(*=======================================================*)
	20:
		IF fb_state_entry.E THEN
			haspel1_ctrl_out.b_init := TRUE;
			haspel2_ctrl_out.b_init := TRUE;
			haspel3_ctrl_out.b_init := TRUE;
			haspel4_ctrl_out.b_init := TRUE;
		END_IF
		(*-----------------------Weiterschaltbedingungen----------------------------*)
		IF  	haspel1_ctrl_in.b_bereit AND
			haspel2_ctrl_in.b_bereit AND
			haspel3_ctrl_in.b_bereit AND
			haspel4_ctrl_in.b_bereit
			THEN
				haspel1_ctrl_out.b_init := FALSE;
				haspel2_ctrl_out.b_init := FALSE;
				haspel3_ctrl_out.b_init := FALSE;
				haspel4_ctrl_out.b_init := FALSE;
				fb_tof_motor.IN := TRUE;
				fb_state_entry.i16_next_step := BEREIT;
		END_IF

(*=======================================================*)
	BEREIT: (* Haspelmotor läuft *)
		IF fb_state_entry.E THEN
			st_ctrl_out.b_bereit := TRUE;
		END_IF

		a_motor_drehrichtung_links 	:= e_druckwaechter AND fb_tof_motor.Q AND b_drehrichtung_antrieb_links;
		a_motor_drehrichtung_rechts := e_druckwaechter AND fb_tof_motor.Q AND NOT b_drehrichtung_antrieb_links;

		(* Abschaltzeit für Haspelmotor nachtriggern*)
		IF 	haspel1_ctrl_in.b_kontroller_start OR
			haspel2_ctrl_in.b_kontroller_start OR
			haspel3_ctrl_in.b_kontroller_start OR
			haspel4_ctrl_in.b_kontroller_start
			THEN
				fb_tof_motor.IN := TRUE;
		ELSE
			fb_tof_motor.IN := FALSE;
		END_IF

(*=======================================================*)
	FEHLER:
		IF fb_state_entry.E THEN
			fb_ton_quitt.IN := FALSE;
			st_ctrl_out.b_fehler := TRUE;
			haspel1_ctrl_out.b_stop := FALSE;
			haspel2_ctrl_out.b_stop := FALSE;
			haspel3_ctrl_out.b_stop := FALSE;
			haspel4_ctrl_out.b_stop := FALSE;
			haspel1_ctrl_out.b_quitt := FALSE;
			haspel2_ctrl_out.b_quitt := FALSE;
			haspel3_ctrl_out.b_quitt := FALSE;
			haspel4_ctrl_out.b_quitt := FALSE;
			a_motor_drehrichtung_links 	:= FALSE;
			a_motor_drehrichtung_rechts := FALSE;
		END_IF

		(*-----------------------Weiterschaltbedingungen----------------------------*)
		IF st_ctrl_in.b_quitt AND NOT fb_state_entry.E THEN
			haspel1_ctrl_out.b_quitt := TRUE;
			haspel2_ctrl_out.b_quitt := TRUE;
			haspel3_ctrl_out.b_quitt := TRUE;
			haspel4_ctrl_out.b_quitt := TRUE;
			st_ctrl_out.b_fehler := FALSE;
			fb_ton_quitt.IN := TRUE;
		END_IF

		IF fb_ton_quitt.Q THEN
			fb_ton_quitt.IN := FALSE;
			fb_state_entry.i16_next_step := INIT;
		END_IF

(*=======================================================*)
	STOP:
		IF fb_state_entry.E THEN
			a_motor_drehrichtung_links 	:= FALSE;
			a_motor_drehrichtung_rechts := FALSE;
			haspel1_ctrl_out.b_stop := TRUE;
			haspel2_ctrl_out.b_stop := TRUE;
			haspel3_ctrl_out.b_stop := TRUE;
			haspel4_ctrl_out.b_stop := TRUE;
			haspel1_ctrl_out.b_quitt := FALSE;
			haspel2_ctrl_out.b_quitt := FALSE;
			haspel3_ctrl_out.b_quitt := FALSE;
			haspel4_ctrl_out.b_quitt := FALSE;
			fb_ton_quitt.IN := FALSE;
		END_IF

		(*-----------------------Weiterschaltbedingungen----------------------------*)
		IF st_ctrl_in.b_quitt AND NOT fb_state_entry.E THEN
			haspel1_ctrl_out.b_stop := FALSE;
			haspel2_ctrl_out.b_stop := FALSE;
			haspel3_ctrl_out.b_stop := FALSE;
			haspel4_ctrl_out.b_stop := FALSE;
			haspel1_ctrl_out.b_quitt := TRUE;
			haspel2_ctrl_out.b_quitt := TRUE;
			haspel3_ctrl_out.b_quitt := TRUE;
			haspel4_ctrl_out.b_quitt := TRUE;

			fb_ton_quitt.IN := TRUE;
		END_IF

		IF fb_ton_quitt.Q THEN
			fb_ton_quitt.IN := FALSE;
			fb_state_entry.i16_next_step := INIT;
		END_IF
END_CASE

fb_state_entry(
	i16_next_step:= , 
	i16_pos:= 2,
	s_debugtext:= ,
	E=> , 
	X=> , 
	i16_step=> ,
	i16_last_step=> );

IF st_config.b_config_fertig THEN
	(* Fehlermeldungen und Betriebsmeldungen ab dem Startindex in die globalen Meldungsarrays schreiben *)
	garr_stoermeldungen[st_config.i16_meld_startindex + 0] := FALSE;
	garr_stoermeldungen[st_config.i16_meld_startindex + 1] := FALSE;
	garr_stoermeldungen[st_config.i16_meld_startindex + 2] := FALSE;
	garr_stoermeldungen[st_config.i16_meld_startindex + 3] := FALSE;
	garr_stoermeldungen[st_config.i16_meld_startindex + 4] := FALSE;
	garr_stoermeldungen[st_config.i16_meld_startindex + 5] := FALSE;
	garr_stoermeldungen[st_config.i16_meld_startindex + 6] := FALSE;
	garr_stoermeldungen[st_config.i16_meld_startindex + 7] := FALSE;
	garr_stoermeldungen[st_config.i16_meld_startindex + 8] := FALSE;
	garr_stoermeldungen[st_config.i16_meld_startindex + 9] := FALSE;
	garr_stoermeldungen[st_config.i16_meld_startindex + 10] := FALSE;
	garr_stoermeldungen[st_config.i16_meld_startindex + 11] := FALSE;
	garr_stoermeldungen[st_config.i16_meld_startindex + 12] := FALSE;
	garr_stoermeldungen[st_config.i16_meld_startindex + 13] := FALSE;
	garr_stoermeldungen[st_config.i16_meld_startindex + 14] := FALSE;
	garr_stoermeldungen[st_config.i16_meld_startindex + 15] := FALSE;
	garr_stoermeldungen[st_config.i16_meld_startindex + 16] := FALSE;
	garr_stoermeldungen[st_config.i16_meld_startindex + 17] := FALSE;
	garr_stoermeldungen[st_config.i16_meld_startindex + 18] := FALSE;
	garr_stoermeldungen[st_config.i16_meld_startindex + 19] := FALSE;
	
	garr_betriebsmeldungen[st_config.i16_meld_startindex + 0] := FALSE;
	garr_betriebsmeldungen[st_config.i16_meld_startindex + 1] := FALSE;
	garr_betriebsmeldungen[st_config.i16_meld_startindex + 2] := FALSE;
	garr_betriebsmeldungen[st_config.i16_meld_startindex + 3] := FALSE;
	garr_betriebsmeldungen[st_config.i16_meld_startindex + 4] := FALSE;
	garr_betriebsmeldungen[st_config.i16_meld_startindex + 5] := FALSE;
	garr_betriebsmeldungen[st_config.i16_meld_startindex + 6] := FALSE;
	garr_betriebsmeldungen[st_config.i16_meld_startindex + 7] := FALSE;
	garr_betriebsmeldungen[st_config.i16_meld_startindex + 8] := FALSE;
	garr_betriebsmeldungen[st_config.i16_meld_startindex + 9] := FALSE;
	garr_betriebsmeldungen[st_config.i16_meld_startindex + 10] := FALSE;
	garr_betriebsmeldungen[st_config.i16_meld_startindex + 11] := FALSE;
	garr_betriebsmeldungen[st_config.i16_meld_startindex + 12] := FALSE;
	garr_betriebsmeldungen[st_config.i16_meld_startindex + 13] := FALSE;
	garr_betriebsmeldungen[st_config.i16_meld_startindex + 14] := FALSE;
	garr_betriebsmeldungen[st_config.i16_meld_startindex + 15] := FALSE;
	garr_betriebsmeldungen[st_config.i16_meld_startindex + 16] := FALSE;
	garr_betriebsmeldungen[st_config.i16_meld_startindex + 17] := FALSE;
	garr_betriebsmeldungen[st_config.i16_meld_startindex + 18] := FALSE;
	garr_betriebsmeldungen[st_config.i16_meld_startindex + 19] := FALSE;
END_IF
END_PROGRAM

(* POU EPT Lib/Programmbausteine/Routing/PC-Suche/ST_RoutingNachbarPC, ST *)
PROGRAM ST_RoutingNachbarPC
VAR_INPUT
	st_config						: struct_config;
	st_ctrl_in						: struct_ctrl_in;
END_VAR
VAR_OUTPUT
	st_ctrl_out					: struct_ctrl_out;
END_VAR
VAR
	arr_read_routing_info			: ARRAY [0..31] OF ST_AmsRouteEntry;
	fb_add_route_entry			: FB_AddRouteEntry;
	fb_enum_route_entry			: FB_EnumRouteEntry;
	fb_ton_quitt					: TON;
	fb_state_entry					: ST_StateEntry;
	i16_geschriebene_eintraege	: INT := 0;
	i16_vorhandene_eintraege		: INT := 0;
	b_ibn_start_routing			: BOOL := FALSE;
	fb_r_trig_ibn_start_routing		: R_TRIG;
	fb_ton_ibn_start_routing		: TON;
	sm_fehler_remotesuche		: BOOL := FALSE;
	sm_fehler_netid				: BOOL := FALSE;
	fb_suche_remote_pc			: ST_SucheRemotePC;
	fb_get_local_ams_netid		: ST_GetLocalAMSNetID;
	i16_eintrag					: INT := 0;
END_VAR
fb_ton_quitt(IN:= , PT:= t#100ms, Q=> , ET=> );
fb_r_trig_ibn_start_routing(CLK:= b_ibn_start_routing, Q=> );
fb_ton_ibn_start_routing(IN:= , PT:= t#1s, Q=> , ET=> );

IF fb_r_trig_ibn_start_routing.Q THEN
	fb_ton_ibn_start_routing.IN := TRUE;
ELSE
	IF fb_ton_ibn_start_routing.Q THEN
		b_ibn_start_routing := FALSE;
	 	fb_ton_ibn_start_routing.IN := FALSE;
	END_IF
END_IF

fb_state_entry(
	i16_next_step:= ,
	i16_pos:= 1,
	s_debugtext:= ,
	E=> ,
	X=> ,
	i16_step=> ,
	i16_last_step=> );

CASE fb_state_entry.i16_step OF
(*=======================================================*)
	0:	(* Initialisierung *)
		st_ctrl_out.b_fehler := TRUE;
		st_ctrl_out.b_bereit := TRUE;
		st_ctrl_out.b_fertig := TRUE;
		fb_add_route_entry.bExecute := FALSE;
		fb_enum_route_entry.bExecute := FALSE;
		fb_suche_remote_pc.bQuit := FALSE;
		fb_suche_remote_pc.bExecute := FALSE;
		fb_get_local_ams_netid .bQuit := FALSE;
		fb_get_local_ams_netid.bExecute := FALSE;
		fb_enum_route_entry.eCmd := eEnumCmd_First;
		i16_geschriebene_eintraege := 0;
		i16_vorhandene_eintraege := 0;
		sm_fehler_remotesuche := FALSE;
		sm_fehler_netid := FALSE;

		FOR i16_eintrag := 0  TO (SIZEOF (arr_read_routing_info) / SIZEOF (arr_read_routing_info[0])) BY 1DO
			arr_read_routing_info[i16_eintrag].sName := '';
			arr_read_routing_info[i16_eintrag].sNetID := '';
			arr_read_routing_info[i16_eintrag].sAddress := '';
			arr_read_routing_info[i16_eintrag].eTransport := eRouteTransport_TCP_IP;
		END_FOR

		fb_state_entry.i16_next_step := 10;

(*=======================================================*)
	10:	(* Die AMS-NetID des lokalen PC ermitteln *)
		IF fb_state_entry.E THEN
			fb_get_local_ams_netid.bExecute := TRUE;
		END_IF

		IF fb_get_local_ams_netid.bBusy THEN
			fb_get_local_ams_netid.bExecute := FALSE;
			fb_state_entry.i16_next_step := 20;
		END_IF

(*=======================================================*)
	20:
		IF NOT fb_get_local_ams_netid.bBusy  THEN
			IF NOT fb_get_local_ams_netid.bError THEN
				fb_state_entry.i16_next_step := 100;
			ELSE	(* Fehler *)
				sm_fehler_netid := TRUE;
				fb_state_entry.i16_next_step := 1000;
			END_IF
		END_IF

(*=======================================================*)
	100:	(* Ersten Routing Eintrag im Routingtable lesen *)
		IF fb_state_entry.E THEN
			fb_enum_route_entry.bExecute := TRUE;
		END_IF

		IF fb_enum_route_entry.bBusy THEN
			fb_enum_route_entry.bExecute := FALSE;
			fb_state_entry.i16_next_step := 110;
		END_IF

(*=======================================================*)
	110:	(* Routinginformation ist vorhanden *)
		IF NOT fb_enum_route_entry.bBusy  THEN
			IF NOT fb_enum_route_entry.bError THEN
				IF NOT fb_enum_route_entry.bEOE THEN
					arr_read_routing_info[i16_vorhandene_eintraege] := fb_enum_route_entry.stRoute;
					fb_enum_route_entry.eCmd := eEnumCmd_Next;
					fb_state_entry.i16_next_step := 120;
				ELSE	(* Alle vorhandenen Routingeinträge  wurden eingelesen*)
					fb_state_entry.i16_next_step := 130;
				END_IF
			ELSE	(* Fehler *)
				fb_state_entry.i16_next_step := 1000;
			END_IF
		END_IF

(*=======================================================*)
	120:	(* Zähler erhöhen *)
		IF fb_state_entry.E THEN
			i16_vorhandene_eintraege := i16_vorhandene_eintraege + 1;
		END_IF

		fb_state_entry.i16_next_step := 100;

(*=======================================================*)
	130:	(* Suche Nachbar-PCs im Maschinennetz *)
		IF fb_state_entry.E THEN
			fb_suche_remote_pc.bExecute := TRUE;
		END_IF

		IF fb_suche_remote_pc.bBusy THEN
			fb_suche_remote_pc.bExecute := FALSE;
			fb_state_entry.i16_next_step := 140;
		END_IF

(*=======================================================*)
	140:	(* Suchvorgang und beendet *)
		IF NOT fb_suche_remote_pc.bBusy  THEN
			IF NOT fb_suche_remote_pc.bError THEN
				fb_state_entry.i16_next_step := 150;
			ELSE	(* Fehler *)
				sm_fehler_remotesuche := TRUE;
				fb_state_entry.i16_next_step := 1000;
			END_IF
		END_IF

(*=======================================================*)
	150:	(* Die Route der gefundenen Nachbar-PCs eintragen *)
		IF fb_state_entry.E THEN
			fb_add_route_entry.stRoute.sName := fb_suche_remote_pc.st_remote_pcinfo_struct[i16_geschriebene_eintraege].Name;
			fb_add_route_entry.stRoute.sNetID := fb_suche_remote_pc.st_remote_pcinfo_struct[i16_geschriebene_eintraege].NetId;
			fb_add_route_entry.stRoute.sAddress := DELETE(fb_add_route_entry.stRoute.sNetID, 4, 12);
			fb_add_route_entry.stRoute.eTransport := eRouteTransport_TCP_IP;
			fb_add_route_entry.bExecute :=TRUE;
			i16_geschriebene_eintraege := i16_geschriebene_eintraege + 1;
		END_IF

		IF fb_add_route_entry.bBusy THEN
			fb_add_route_entry.bExecute := FALSE;
			fb_state_entry.i16_next_step := 160;
		END_IF

(*=======================================================*)
	160:	(* Routingtable füllen läuft *)
		IF NOT fb_add_route_entry.bBusy THEN
			IF NOT fb_add_route_entry.bError THEN	(* Route wurde erfolgreich hinzugefügt *)
				(* Routingtable mit fehlenden Stationsadressen füllen wenn notwendig *)
				IF i16_geschriebene_eintraege < i16_vorhandene_eintraege THEN
					fb_state_entry.i16_next_step := 150;
				ELSE
					fb_state_entry.i16_next_step := 999;
				END_IF
			ELSE	(* Fehler *)
				fb_state_entry.i16_next_step := 1000;
			END_IF
		END_IF

(*=======================================================*)
	999: (* Ende: Alle Stationen wurden im Routingtable eingetragen *)
		IF fb_state_entry.E THEN
			st_ctrl_out.b_fertig := TRUE;
		END_IF

(*=======================================================*)
	1000: (* Fehler *)
		IF fb_state_entry.E THEN
			st_ctrl_out.b_fehler := TRUE;
			fb_ton_quitt.IN := FALSE;
			fb_add_route_entry.bExecute := FALSE;
			fb_enum_route_entry.bExecute := FALSE;
			fb_suche_remote_pc.bExecute := FALSE;
			fb_suche_remote_pc.bQuit := FALSE;
			fb_get_local_ams_netid.bExecute := FALSE;
			fb_get_local_ams_netid.bQuit := FALSE;
		END_IF

		(*-----------------------Weiterschaltbedingungen----------------------------*)
		IF st_ctrl_in.b_quitt AND NOT fb_state_entry.E THEN
			st_ctrl_out.b_fehler := FALSE;
			fb_ton_quitt.IN := TRUE;
			fb_suche_remote_pc.bQuit := TRUE;
			fb_get_local_ams_netid .bQuit := TRUE;
		END_IF

		IF fb_ton_quitt.Q OR  fb_r_trig_ibn_start_routing.Q THEN
			fb_ton_quitt.IN := FALSE;
			fb_state_entry.i16_next_step := 0;
		END_IF
END_CASE

fb_state_entry(
	i16_next_step:= , 
	i16_pos:= 2,
	s_debugtext:= ,
	E=> ,
	X=> , 
	i16_step=> ,
	i16_last_step=> );

fb_get_local_ams_netid(
	bExecute:= , 
	bQuit:= , 
	bBusy=> , 
	bReady=> , 
	bError=> , 
	nErrId=> , 
	s_ams_netid=> );

fb_suche_remote_pc(
	bExecute:= ,
	bQuit:= , 
	bBusy=> , 
	bError=> , 
	nErrId=> );

fb_add_route_entry(
	sNetID:= ,
	stRoute:= ,
	bExecute:= ,
	tTimeout:= DEFAULT_ADS_TIMEOUT,
	bBusy=> , 
	bError=> , 
	nErrID=> );

fb_enum_route_entry(
	sNetID:= ,
	eCmd:= , 
	bExecute:= , 
	tTimeout:= DEFAULT_ADS_TIMEOUT,
	bBusy=> , 
	bError=> , 
	nErrID=> , 
	bEOE=> , 
	stRoute=> );

IF st_config.b_config_fertig THEN
	garr_stoermeldungen[st_config.i16_meld_startindex + 0] := sm_fehler_remotesuche;
	garr_stoermeldungen[st_config.i16_meld_startindex + 1] := sm_fehler_netid;
	garr_stoermeldungen[st_config.i16_meld_startindex + 2] := FALSE;
	garr_stoermeldungen[st_config.i16_meld_startindex + 3] := FALSE;
	garr_stoermeldungen[st_config.i16_meld_startindex + 4] := FALSE;
	garr_stoermeldungen[st_config.i16_meld_startindex + 5] := FALSE;
	garr_stoermeldungen[st_config.i16_meld_startindex + 6] := FALSE;
	garr_stoermeldungen[st_config.i16_meld_startindex + 7] := FALSE;
	garr_stoermeldungen[st_config.i16_meld_startindex + 8] := FALSE;
	garr_stoermeldungen[st_config.i16_meld_startindex + 9] := FALSE;
	garr_stoermeldungen[st_config.i16_meld_startindex + 10] := FALSE;
	garr_stoermeldungen[st_config.i16_meld_startindex + 11] := FALSE;
	garr_stoermeldungen[st_config.i16_meld_startindex + 12] := FALSE;
	garr_stoermeldungen[st_config.i16_meld_startindex + 13] := FALSE;
	garr_stoermeldungen[st_config.i16_meld_startindex + 14] := FALSE;
	garr_stoermeldungen[st_config.i16_meld_startindex + 15] := FALSE;
	garr_stoermeldungen[st_config.i16_meld_startindex + 16] := FALSE;
	garr_stoermeldungen[st_config.i16_meld_startindex + 17] := FALSE;
	garr_stoermeldungen[st_config.i16_meld_startindex + 18] := FALSE;
	garr_stoermeldungen[st_config.i16_meld_startindex + 19] := FALSE;
	
	garr_betriebsmeldungen[st_config.i16_meld_startindex + 0] := FALSE;
	garr_betriebsmeldungen[st_config.i16_meld_startindex + 1] := FALSE;
	garr_betriebsmeldungen[st_config.i16_meld_startindex + 2] := FALSE;
	garr_betriebsmeldungen[st_config.i16_meld_startindex + 3] := FALSE;
	garr_betriebsmeldungen[st_config.i16_meld_startindex + 4] := FALSE;
	garr_betriebsmeldungen[st_config.i16_meld_startindex + 5] := FALSE;
	garr_betriebsmeldungen[st_config.i16_meld_startindex + 6] := FALSE;
	garr_betriebsmeldungen[st_config.i16_meld_startindex + 7] := FALSE;
	garr_betriebsmeldungen[st_config.i16_meld_startindex + 8] := FALSE;
	garr_betriebsmeldungen[st_config.i16_meld_startindex + 9] := FALSE;
	garr_betriebsmeldungen[st_config.i16_meld_startindex + 10] := FALSE;
	garr_betriebsmeldungen[st_config.i16_meld_startindex + 11] := FALSE;
	garr_betriebsmeldungen[st_config.i16_meld_startindex + 12] := FALSE;
	garr_betriebsmeldungen[st_config.i16_meld_startindex + 13] := FALSE;
	garr_betriebsmeldungen[st_config.i16_meld_startindex + 14] := FALSE;
	garr_betriebsmeldungen[st_config.i16_meld_startindex + 15] := FALSE;
	garr_betriebsmeldungen[st_config.i16_meld_startindex + 16] := FALSE;
	garr_betriebsmeldungen[st_config.i16_meld_startindex + 17] := FALSE;
	garr_betriebsmeldungen[st_config.i16_meld_startindex + 18] := FALSE;
	garr_betriebsmeldungen[st_config.i16_meld_startindex + 19] := FALSE;
END_IF
END_PROGRAM

(* POU EPT Lib/Programmbausteine/Routing/PC-Suche/ST_SucheRemotePC, ST *)
FUNCTION_BLOCK ST_SucheRemotePC
VAR_INPUT
	bExecute			: BOOL;
	bQuit				: BOOL;
END_VAR
VAR_OUTPUT
	bBusy				: BOOL;
	bError				: BOOL;
	nErrId				: UDINT;
END_VAR
VAR
	fb_ton_quitt					: TON;
	fb_state_entry					: ST_StateEntry;
	fb_r_trig_execute				: R_TRIG;
	i							: INT := 0;
	b_ibn_start					: BOOL := FALSE;
	fb_r_trig_ibn_start				: R_TRIG;
	fb_ton_ibn_start				: TON;
	fb_get_remote_pcinfo			:GetRemotePCInfo;
	st_remote_pcinfo_struct		:REMOTEPCINFOSTRUCT;
							       (*TYPE REMOTEPCINFOSTRUCT
									ARRAY[0..99] OF REMOTEPC;
								END_TYPE*)
							      (*TYPE REMOTEPC
								STRUCT
									NetId 	: T_AmsNetId;
									Name 	: STRING(31);
								END_STRUCT
								END_TYPE*)
END_VAR
fb_r_trig_execute(CLK:= bExecute, Q=> );
fb_ton_quitt(IN:= , PT:= t#100ms, Q=> , ET=> );

fb_r_trig_ibn_start(CLK:= b_ibn_start, Q=> );
fb_ton_ibn_start(IN:= , PT:= t#1s, Q=> , ET=> );

IF fb_r_trig_ibn_start.Q THEN
	fb_ton_ibn_start.IN := TRUE;
ELSE
	IF fb_ton_ibn_start.Q THEN
		b_ibn_start := FALSE;
	 	fb_ton_ibn_start.IN := FALSE;
	END_IF
END_IF

fb_state_entry(
	i16_next_step:= ,
	i16_pos:= 1,
	s_debugtext:= ,
	E=> ,
	X=> , 
	i16_step=> ,
	i16_last_step=> );

CASE fb_state_entry.i16_step OF
(*=======================================================*)
	0:(* INIT *)
		bBusy := FALSE;
		bError := FALSE;
		nErrId := 0;
		fb_get_remote_pcinfo.START := FALSE;
		fb_state_entry.i16_next_step := 10;

(*=======================================================*)
	10:	(* Warte auf Execute-Befehl *)
		IF fb_state_entry.E THEN
			bBusy := FALSE;
		END_IF

		IF fb_r_trig_execute.Q OR fb_r_trig_ibn_start.Q THEN
			bBusy := TRUE;
			fb_state_entry.i16_next_step := 100;
		END_IF

(*=======================================================*)
	100:	(* Starte mit Auslesen der über ADS verbundenen Nachbar-PCs *)
		IF fb_state_entry.E THEN
			fb_get_remote_pcinfo.START := TRUE;
		END_IF

		IF fb_get_remote_pcinfo.BUSY THEN
			fb_get_remote_pcinfo.START := FALSE;
			fb_state_entry.i16_next_step := 110;
		END_IF

(*=======================================================*)
	110:	(* Routinginformation über die Nachbar-PCs ist vorhanden *)
		IF NOT fb_get_remote_pcinfo.BUSY  THEN
			IF NOT fb_get_remote_pcinfo.ERR THEN
				fb_state_entry.i16_next_step := 999;
			ELSE	(* Fehler *)
				fb_state_entry.i16_next_step := 1000;
			END_IF
		END_IF

(*=======================================================*)
	999:	(* Kontrollschritt: Nachbar-PC ist gefunden *)
		fb_state_entry.i16_next_step := 10;

(*=======================================================*)
	1000: (* Fehler *)
		IF fb_state_entry.E THEN
			bBusy := FALSE;
			bError := TRUE;
			fb_ton_quitt.IN := FALSE;
		END_IF

		(*-----------------------Weiterschaltbedingungen----------------------------*)
		IF bQuit AND NOT fb_state_entry.E THEN
			bError := FALSE;
			fb_ton_quitt.IN := TRUE;
		END_IF

		IF fb_ton_quitt.Q THEN
			fb_ton_quitt.IN := FALSE;
			fb_state_entry.i16_next_step := 0;
		END_IF
END_CASE

fb_state_entry(
	i16_next_step:= , 
	i16_pos:= 2,
	s_debugtext:= ,
	E=> ,
	X=> , 
	i16_step=> ,
	i16_last_step=> );

fb_get_remote_pcinfo(
	NETID:= , 
	START:= , 
	TMOUT:= , 
	BUSY=> , 
	ERR=> , 
	ERRID=> , 
	RemotePCInfo=> st_remote_pcinfo_struct);
END_FUNCTION_BLOCK

(* POU EPT Lib/Funktionen/BOOLARRAY_TO_BYTE, ST *)
FUNCTION BOOLARRAY_TO_BYTE : BYTE
VAR_INPUT
	p_adr_buffer			: POINTER TO ARRAY[0..7] OF BOOL;
END_VAR
VAR
	tmp_buffer			: ARRAY[0..7] OF BOOL;
	tmp_byte				: BYTE;
	i16_index			: INT;
END_VAR
(* Aus einem Boolarray, soll ein Byte entstehen *)
tmp_buffer := p_adr_buffer^;

tmp_byte := 2#0;

FOR i16_index := 7 TO 0 BY -1 DO
	tmp_byte := tmp_byte OR BOOL_TO_BYTE(tmp_buffer[i16_index]);
	IF i16_index > 0 THEN
		tmp_byte := SHL(tmp_byte, 1);
	END_IF
END_FOR;

BOOLARRAY_TO_BYTE := tmp_byte; (* Rückgabewert der Funktion *)
END_FUNCTION

(* POU EPT Lib/Funktionen/BOOLARRAY_TO_DWORD, ST *)
FUNCTION BOOLARRAY_TO_DWORD : DWORD
VAR_INPUT
	p_adr_buffer			: POINTER TO ARRAY[0..31] OF BOOL;
END_VAR
VAR
	tmp_buffer			: ARRAY[0..31] OF BOOL;
	tmp_dword			: DWORD;
	i16_index			: INT;
END_VAR
(* Aus einem Boolarray, soll ein Doppelword entstehen *)
tmp_buffer := p_adr_buffer^;

tmp_dword := 2#0;

FOR i16_index := 31 TO 0 BY -1 DO
	tmp_dword := tmp_dword OR BOOL_TO_DWORD(tmp_buffer[i16_index]);
	IF i16_index > 0 THEN
		tmp_dword := SHL(tmp_dword, 1);
	END_IF
END_FOR;

BOOLARRAY_TO_DWORD := tmp_dword; (* Rückgabewert der Funktion *)
END_FUNCTION

(* POU EPT Lib/Funktionen/BOOLARRAY_TO_WORD, ST *)
FUNCTION BOOLARRAY_TO_WORD : WORD
VAR_INPUT
	p_adr_buffer			: POINTER TO ARRAY[0..15] OF BOOL;
END_VAR
VAR
	tmp_buffer			: ARRAY[0..15] OF BOOL;
	tmp_word			: WORD;
	i16_index			: INT;
END_VAR
(* Aus einem Boolarray, soll ein Word entstehen *)
tmp_buffer := p_adr_buffer^;

tmp_word := 2#0;

FOR i16_index := 15 TO 0 BY -1 DO
	tmp_word := tmp_word OR BOOL_TO_WORD(tmp_buffer[i16_index]);
	IF i16_index > 0 THEN
		tmp_word := SHL(tmp_word, 1);
	END_IF
END_FOR;

BOOLARRAY_TO_WORD := tmp_word; (* Rückgabewert der Funktion *)
END_FUNCTION

(* POU EPT Lib/Funktionen/BYTEARRAY_TO_STRING_WITH_DELIMITER, ST *)
FUNCTION BYTEARRAY_TO_STRING_WITH_DELIMITER : STRING
VAR_INPUT
	p_adr_buffer			: POINTER TO ARRAY[0..100] OF BYTE;
	i16_buffer_laenge		: INT;
	str_delimiter			: STRING; (* Punkt zum trennen der einzelnen Zahlen in der Net-Adresse *)
END_VAR
VAR
	tmp_buffer			: ARRAY[0..100] OF BYTE;
	tmp_string			: STRING;
	i16_index			: INT;
END_VAR
(* Aus einem Bytearray, welches die einzelnen Zahlen der Net-Adresse beinhaltet wird ein String erzeugt, welcher die Zahlen getrennt durch Punkte enthält *)
tmp_buffer := p_adr_buffer^;

tmp_string := ''; (* leerer String *)
FOR i16_index := 0 TO i16_buffer_laenge - 1 DO
	tmp_string :=CONCAT(tmp_string ,BYTE_TO_STRING(tmp_buffer[i16_index]));
	IF i16_index < i16_buffer_laenge - 1 THEN
		tmp_string := CONCAT(tmp_string,str_delimiter); (* "Punkt" einfügen in den String *)
	END_IF;
END_FOR;

BYTEARRAY_TO_STRING_WITH_DELIMITER := tmp_string; (* Rückgabewert der Funktion *)
END_FUNCTION

(* POU EPT Lib/Funktionen/Checks/CheckBounds, ST *)
FUNCTION CheckBounds : DINT
VAR_INPUT
	index, lower, upper 	: DINT;
END_VAR
VAR
END_VAR
IF index<lower THEN
	CheckBounds_ErrCnt := CheckBounds_ErrCnt + 1;
	CheckBounds := lower;
ELSIF index>upper THEN
	CheckBounds_ErrCnt := CheckBounds_ErrCnt + 1;
	CheckBounds := upper;
ELSE
	CheckBounds := index;
END_IF
END_FUNCTION

(* POU EPT Lib/Funktionen/Checks/CheckDivByte, ST *)
FUNCTION CheckDivByte : BYTE
VAR_INPUT
	divisor			 	: BYTE;
END_VAR
VAR
END_VAR
IF divisor = 0 THEN
	CheckByteZeroDiv_ErrCnt := CheckByteZeroDiv_ErrCnt + 1;
	CheckDivByte := 1;
ELSE
	CheckDivByte := divisor;
END_IF
END_FUNCTION

(* POU EPT Lib/Funktionen/Checks/CheckDivDWord, ST *)
FUNCTION CheckDivDWord : DWORD
VAR_INPUT
	divisor				: DWORD;
END_VAR
VAR
END_VAR
IF divisor = 0 THEN
	CheckDWordZeroDiv_ErrCnt := CheckDWordZeroDiv_ErrCnt + 1;
	CheckDivDWord := 1;
ELSE
	CheckDivDWord := divisor;
END_IF
END_FUNCTION

(* POU EPT Lib/Funktionen/Checks/CheckDivReal, ST *)
FUNCTION CheckDivReal : REAL
VAR_INPUT
	divisor		 		: REAL;
END_VAR
VAR
END_VAR
IF divisor = 0 THEN
	CheckRealZeroDiv_ErrCnt := CheckRealZeroDiv_ErrCnt + 1;
	CheckDivReal := 1;
ELSE
	CheckDivReal := divisor;
END_IF
END_FUNCTION

(* POU EPT Lib/Funktionen/Checks/CheckDivWord, ST *)
FUNCTION CheckDivWord : WORD
VAR_INPUT
	divisor				: WORD;
END_VAR
VAR
END_VAR
IF divisor = 0 THEN
	CheckWordZeroDiv_ErrCnt:= CheckWordZeroDiv_ErrCnt + 1;
	CheckDivWord := 1;
ELSE
	CheckDivWord := divisor;
END_IF
END_FUNCTION

(* POU EPT Lib/Funktionen/Checks/CheckRangeSigned, ST *)
FUNCTION CheckRangeSigned : DINT
VAR_INPUT
    value, lower, upper: DINT;
END_VAR
VAR
END_VAR
IF (value < lower) THEN
	CheckRangeSigned_ErrCnt := CheckRangeSigned_ErrCnt + 1;
	CheckRangeSigned := lower;
ELSIF(value > upper) THEN
	CheckRangeSigned_ErrCnt := CheckRangeSigned_ErrCnt + 1;
	CheckRangeSigned := upper;
ELSE
	CheckRangeSigned := value;
END_IF
END_FUNCTION

(* POU EPT Lib/Funktionen/Checks/CheckRangeUnsigned, ST *)
FUNCTION CheckRangeUnsigned : UDINT
VAR_INPUT
    value, lower, upper: UDINT;
END_VAR
VAR
END_VAR
IF (value < lower) THEN
	CheckRangeUnSigned_ErrCnt := CheckRangeUnsigned_ErrCnt + 1;
	CheckRangeUnsigned := lower;
ELSIF(value > upper) THEN
	CheckRangeUnsigned_ErrCnt := CheckRangeUnsigned_ErrCnt + 1;
	CheckRangeUnsigned := upper;
ELSE
	CheckRangeUnsigned := value;
END_IF
END_FUNCTION

(* POU EPT Lib/Funktionen/F_rSign, ST *)
FUNCTION F_rSign : LREAL
VAR_INPUT
	rValue		:LREAL;	(*Zahl*)
END_VAR
IF rValue >= 0 THEN
	F_rSign := 1;
ELSE
	F_rSign := -1;
END_IF
END_FUNCTION

(* POU EPT Lib/Funktionen/F_Vergleich_Real, ST *)
FUNCTION F_Vergleich_Real : BOOL
VAR_INPUT
	r_wert			: REAL;
	r_vergleichswert	: REAL;
END_VAR
VAR
	r_toleranz		: REAL := 0.001;
END_VAR
IF ABS(r_wert - r_vergleichswert) < r_toleranz THEN
	F_Vergleich_Real := TRUE;
ELSE
	F_Vergleich_Real := FALSE;
END_IF
END_FUNCTION

(* POU Gemeinsamkeiten17xx/XML Server/FB_2OrdnerMitDateiErstellen, ST *)
FUNCTION_BLOCK FB_2OrdnerMitDateiErstellen
VAR_INPUT
	bExecute					: BOOL;
	bQuit						: BOOL;
	s_path						: STRING;
	s_dateiname					: STRING;
	s_datei_erweiterung			: STRING;
	s_x_path_name				: STRING;
	s_symname					: STRING;
END_VAR
VAR_IN_OUT
END_VAR
VAR_OUTPUT
	bBusy						: BOOL;
	bError						: BOOL;
	nErrId						: UDINT;

END_VAR
VAR
	fb_enum_find_file_list			: FB_EnumFindFileList;
	fb_enum_find_file_entry			: FB_EnumFindFileEntry;
	fb_create_directory			: FB_CreateDir;	(* mit diesem FB kan nur eine Ordnerverzeichnissstruktur angelegt werden, jedoch keine Dateien erzeugt werden *)
	fb_file_open					: FB_FileOpen;	(* Eine vorhandene Datei öffnen oder eine Neue erzeugen *)
	fb_file_close					: FB_FileClose;
	fb_file_write					: FB_FileWrite;
	h_filehandle					: UINT := 0;(* file handle of the file *)
	arr_file_list					: ARRAY[0..63] OF ST_FindFileEntry;
	fb_ton_quitt					: TON;
	fb_r_trig_execute				: R_TRIG;
	fb_state_entry					: ST_StateEntry;
	temp_string					: STRING[255];
	i16_file_entry_zaehler			: INT := 0;
	i16_file_nr					: INT := 0;
	i							: INT := 0;
	b_pfad_vorhanden			: BOOL;
	b_datei_vorhanden			: BOOL;
	arr_rootpath					: ARRAY[0..2] OF STRING;
END_VAR
fb_r_trig_execute(CLK:= bExecute, Q=> );
fb_ton_quitt(IN:= , PT:= t#100ms, Q=> , ET=> );

(* ======================================Schrittkette======================================== *)
fb_state_entry(
	i16_next_step:= ,
	i16_pos:= 1,
	s_debugtext:= ,
	E=> ,
	X=> ,
	i16_step=> ,
	i16_last_step=> );

CASE fb_state_entry.i16_step OF
(*=======================================================*)
	0:(* INIT *)
		bBusy := FALSE;
		bError := FALSE;
		nErrId := 0;
		fb_create_directory.bExecute := FALSE;
		fb_enum_find_file_list.bExecute := FALSE;
		fb_enum_find_file_entry.bExecute := FALSE;
		fb_file_open.bExecute := FALSE;
		fb_file_close.bExecute := FALSE;
		fb_state_entry.i16_next_step := 10;

(*=======================================================*)
	10:	(* Warte auf Execute-Befehl *)
		IF fb_state_entry.E THEN
			bBusy := FALSE;
		END_IF

		IF fb_r_trig_execute.Q THEN
			bBusy := TRUE;
			b_pfad_vorhanden := FALSE;
			b_datei_vorhanden := FALSE;
			arr_rootpath[0] := MID(s_path, 1,3);
			arr_rootpath[1] := MID(s_path, 4,3);
			arr_rootpath[2] := MID(s_path, 10,3);
			fb_state_entry.i16_next_step := 20;
		END_IF

(*=======================================================*)
	20:	(* Prüfe, ob gewünschter Pfad auf dem Maschinen-PC vorhanden ist *)
		IF fb_state_entry.E THEN
			fb_enum_find_file_list.sPathName := s_path;
			fb_enum_find_file_list.eCmd := eEnumCmd_First;
			fb_enum_find_file_list.bExecute := TRUE;
		END_IF

		IF fb_enum_find_file_list.bBusy THEN
			fb_enum_find_file_list.bExecute := FALSE;
			fb_state_entry.i16_next_step := 30;
		END_IF

(*=======================================================*)
	30:	(* Auswerten des Ordner-Suchergebnis *)
		IF NOT fb_enum_find_file_list.bBusy THEN
			fb_enum_find_file_list.bExecute := FALSE;
		 	IF fb_enum_find_file_list.bError OR fb_enum_find_file_list.bEOE THEN
				 IF fb_enum_find_file_list.nFindFiles=0 THEN
					b_pfad_vorhanden := FALSE;
					fb_state_entry.i16_next_step := 40;	(* Pfad nicht vorhanden -> wird angelegt *)
				ELSE
					b_pfad_vorhanden := TRUE;
					fb_state_entry.i16_next_step := 60;	(* O.K. Pfad vorhanden -> Datei prüfen *)
				END_IF
			END_IF
		END_IF

(*=======================================================*)
	40:	(* Erstellen des ersten Ordnerverzeichnisses auf dem Laufwerk des Maschinen-PCs *)
		IF fb_state_entry.E THEN
			fb_create_directory.sPathName := s_path;
			fb_create_directory.bExecute := TRUE;
		END_IF

		IF fb_create_directory.bBusy THEN
			fb_create_directory.bExecute := FALSE;
			fb_state_entry.i16_next_step := 50;
		END_IF

(*=======================================================*)
	50:	(* Ordner wurde erstellt *)
		IF NOT fb_create_directory.bBusy  THEN
			IF NOT fb_create_directory.bError THEN
				fb_state_entry.i16_next_step := 60;	(* Ordnerverzeichnis wurde erfolgreich erstellt -> eine neue Datei anlegen oder eine Vorhandene öffnen *)
			ELSE
				fb_state_entry.i16_next_step := 1000;	(* Fehler *)
			END_IF
		END_IF

(*=======================================================*)
	60:	(* Prüfe, ob die gewünschte Datei in diesem Ordnerverzeichnis vorhanden ist *)
		IF fb_state_entry.E THEN
			temp_string := '';
			temp_string := CONCAT(temp_string, s_path);
			temp_string := CONCAT(temp_string, '\');
			temp_string := CONCAT(temp_string, s_dateiname);
			temp_string := CONCAT(temp_string, s_datei_erweiterung);
			fb_enum_find_file_entry.sPathName := temp_string;
			fb_enum_find_file_entry.eCmd := eEnumCmd_First;
			fb_enum_find_file_entry.bExecute := TRUE;
		END_IF

		IF fb_enum_find_file_entry.bBusy THEN
			fb_enum_find_file_entry.bExecute := FALSE;
			fb_state_entry.i16_next_step := 70;
		END_IF

(*=======================================================*)
	70:	(* Auswerten des Datei-Suchergebnis *)
		IF NOT fb_enum_find_file_entry.bBusy THEN
			fb_enum_find_file_entry.bExecute := FALSE;
		 	IF NOT fb_enum_find_file_entry.bError THEN
				IF fb_enum_find_file_entry.bEOE THEN
					IF fb_enum_find_file_entry.stFindFile.sFileName = CONCAT(s_dateiname, s_datei_erweiterung) THEN
					(* Datei bereits vorhanden *)
						b_datei_vorhanden := TRUE;
						fb_state_entry.i16_next_step := 0;
					ELSE
					(* Ende der Fileliste wurde erreicht und die gesuchte Datei ist  nicht vorhanden -> muss später angelegt werden *)
						b_datei_vorhanden := FALSE;
						fb_state_entry.i16_next_step := 100;
					END_IF
				ELSE
				(* Dateisuche im FB mit Abort korrekt beenden *)
					IF fb_enum_find_file_entry.stFindFile.sFileName = CONCAT(s_dateiname, s_datei_erweiterung) THEN
					(* Die gesuchte Datei wurde in der Fileliste gefunden *)
						b_datei_vorhanden := TRUE;
						fb_state_entry.i16_next_step := 80;
					ELSE
					(* Datei ist  nicht vorhanden -> muss später angelegt werden *)
						b_datei_vorhanden := FALSE;
						fb_state_entry.i16_next_step := 80;
					END_IF
				END_IF
			ELSE
				fb_state_entry.i16_next_step := FEHLER;
			END_IF
		END_IF

(*=======================================================*)
	80:	(* Dateisuchen wird beendet *)
		IF fb_state_entry.E THEN
			fb_enum_find_file_entry.eCmd := eEnumCmd_Abort;
			fb_enum_find_file_entry.bExecute := TRUE;
		END_IF

		IF fb_enum_find_file_entry.bBusy THEN
			fb_enum_find_file_entry.bExecute := FALSE;
			fb_state_entry.i16_next_step := 90;
		END_IF

(*=======================================================*)
	90:	(* Filehandle wieder frei *)
		IF NOT fb_enum_find_file_entry.bBusy THEN
			fb_enum_find_file_entry.bExecute := FALSE;
		 	IF NOT fb_enum_find_file_entry.bError AND fb_enum_find_file_entry.bEOE THEN
				fb_state_entry.i16_next_step := 100;
			ELSE
				fb_state_entry.i16_next_step := FEHLER;
			END_IF
		END_IF

(*=======================================================*)
	100:	(* Abfrage auf Datei anlegen *)
		IF fb_state_entry.E THEN
			IF NOT b_datei_vorhanden THEN
				fb_state_entry.i16_next_step := 110;
			ELSE
				fb_state_entry.i16_next_step := 0;	(* Fertig *)
			END_IF
		END_IF

(*=======================================================*)
	110:	(* Erzeugen einer neuen Datei *)
		IF fb_state_entry.E THEN
			temp_string := '';
			temp_string := CONCAT(temp_string, s_path);
			temp_string := CONCAT(temp_string, '\');
			temp_string := CONCAT(temp_string, s_dateiname);
			temp_string := CONCAT(temp_string, s_datei_erweiterung);
			fb_file_open.sPathName := temp_string;
			fb_file_open.nMode := FOPEN_MODEWRITE OR FOPEN_MODEBINARY;
			fb_file_open.bExecute := TRUE;
		END_IF

		IF fb_file_open.bBusy THEN
			fb_file_open.bExecute := FALSE;
			fb_state_entry.i16_next_step := 120;
		END_IF

(*=======================================================*)
	120:	(* Warte bis Datei geöffnet wurde *)
		IF NOT fb_file_open.bBusy  THEN
			IF NOT fb_file_open.bError THEN
				h_filehandle := fb_file_open.hFile;
				fb_state_entry.i16_next_step := 130;
			ELSE	(* Fehler *)
				nErrId := fb_file_open.nErrId;
				fb_state_entry.i16_next_step := 1000;
			END_IF
		END_IF

(*=======================================================*)
	130:	(* Schreibe die Dateistruktur im XML-Format: z.B.*)
		(*
		<Maschine1700_Datensicherung>
		<gst_datensatz>
		</gst_datensatz>
		</Maschine1700_Datensicherung>
		*)
		IF fb_state_entry.E THEN
			temp_string := '';
			temp_string := CONCAT(temp_string, '<');
			temp_string := CONCAT(temp_string, s_x_path_name);
			temp_string := CONCAT(temp_string, '>');
			temp_string := CONCAT(temp_string, '$r$n');

			(* Die Variable "s_xml_variablenname" wird hier schon mit angelegt, *)
			(* damit später beim "WECHSELN>" daraus gelesen werden kann, obwohl noch nichts drin steht *)
			temp_string := CONCAT(temp_string, '<');
			temp_string := CONCAT(temp_string, s_symname);
			temp_string := CONCAT(temp_string, '>');
			temp_string := CONCAT(temp_string, '$r$n');
			temp_string := CONCAT(temp_string, '<');
			temp_string := CONCAT(temp_string, '/');
			temp_string := CONCAT(temp_string, s_symname);
			temp_string := CONCAT(temp_string, '>');
			temp_string := CONCAT(temp_string, '$r$n');

			temp_string := CONCAT(temp_string, '<');
			temp_string := CONCAT(temp_string, '/');
			temp_string := CONCAT(temp_string, s_x_path_name);
			temp_string := CONCAT(temp_string, '>');
			fb_file_write.hFile := h_filehandle;
 			fb_file_write.bExecute := TRUE;
		END_IF

		IF fb_file_write.bBusy THEN
			fb_file_write.bExecute := FALSE;
			fb_state_entry.i16_next_step := 140;
		END_IF

(*=======================================================*)
	140:	(* Warte bis Datei geschrieben wurde *)
		IF NOT fb_file_write.bBusy  THEN
			IF NOT fb_file_write.bError THEN
				fb_state_entry.i16_next_step := 150;
			ELSE	(* Fehler *)
				nErrId := fb_file_write.nErrId;
				fb_state_entry.i16_next_step := 1000;
			END_IF
		END_IF

(*=======================================================*)
	150:	(* Schliesse Datei wieder, damit ein erneuter Zugriff möglich ist *)
		IF fb_state_entry.E THEN
			fb_file_close.hFile := h_filehandle;
			fb_file_close.bExecute := TRUE;
		END_IF

		IF fb_file_close.bBusy THEN
			fb_file_close.bExecute := FALSE;
			fb_state_entry.i16_next_step := 160;
		END_IF

(*=======================================================*)
	160:	(* Warte bis geschlossen *)
		IF NOT fb_file_close.bBusy  THEN
			IF NOT fb_file_close.bError THEN
				h_filehandle := 0;
				fb_state_entry.i16_next_step :=0;
			ELSE	(* Fehler *)
				nErrId := fb_file_close.nErrId;
				fb_state_entry.i16_next_step := 1000;
			END_IF
		END_IF

(*=======================================================*)
	1000: (* Fehler *)
		IF fb_state_entry.E THEN
			bBusy := FALSE;
			bError := TRUE;
			fb_ton_quitt.IN := FALSE;
		END_IF

		(*-----------------------Weiterschaltbedingungen----------------------------*)
		IF bQuit AND NOT fb_state_entry.E THEN
			bError := FALSE;
			fb_ton_quitt.IN := TRUE;
		END_IF

		IF fb_ton_quitt.Q THEN
			fb_ton_quitt.IN := FALSE;
			fb_state_entry.i16_next_step := 0;
		END_IF
END_CASE

fb_state_entry(
	i16_next_step:= , 
	i16_pos:= 2,
	s_debugtext:= ,
	E=> , 
	X=> , 
	i16_step=> ,
	i16_last_step=> );

fb_enum_find_file_list(
	sNetId:= '',
	sPathName:= ,
	eCmd:= ,
	pFindList:= ADR(arr_file_list),
	cbFindList:= SIZEOF(arr_file_list),
	bExecute:= ,
	tTimeout:= DEFAULT_ADS_TIMEOUT,
	bBusy=> ,
	bError=> ,
	nErrID=> , 
	bEOE=> ,
	nFindFiles=> );

fb_enum_find_file_entry(
	sNetId:= '',
	sPathName:= , 
	eCmd:= , 
	bExecute:= , 
	tTimeout:= DEFAULT_ADS_TIMEOUT,
	bBusy=> , 
	bError=> ,
	nErrID=> , 
	bEOE=> , 
	stFindFile=> );

fb_create_directory(
	sNetId:= '',
	sPathName:= ,
	ePath:= PATH_GENERIC,
	bExecute:= ,
	tTimeout:= DEFAULT_ADS_TIMEOUT,
	bBusy=> , 
	bError=> ,
	nErrId=> );

fb_file_open(
	sNetId:= '',
	sPathName:= , 
	nMode:= ,
	ePath:= PATH_GENERIC,
	bExecute:= , 
	tTimeout:= DEFAULT_ADS_TIMEOUT,
	bBusy=> , 
	bError=> , 
	nErrId=> , 
	hFile=> );

fb_file_close(
	sNetId:= '',
	hFile:= , 
	bExecute:= , 
	tTimeout:= t#10s,
	bBusy=> ,
	bError=> ,
	nErrId=> );

fb_file_write(
	sNetId:= '',
	hFile:= , 
	pWriteBuff:= ADR(temp_string),
	cbWriteLen:= LEN(temp_string),
	bExecute:= , 
	tTimeout:= t#10s,
	bBusy=> ,
	bError=> , 
	nErrId=> , 
	cbWrite=> );
END_FUNCTION_BLOCK

(* POU Gemeinsamkeiten17xx/XML Server/FB_Datei_erstellen, ST *)
FUNCTION_BLOCK FB_Datei_erstellen
VAR_INPUT
	bExecute					: BOOL;
	bQuit						: BOOL;
	s_path						: STRING;
	s_dateiname					: STRING;
	s_datei_erweiterung			: STRING;
	s_x_path_name				: STRING;
	s_symname					: STRING;
END_VAR
VAR_IN_OUT
END_VAR
VAR_OUTPUT
	bBusy						: BOOL;
	bError						: BOOL;
	nErrId						: UDINT;
END_VAR
VAR
	fb_enum_find_file_list			: FB_EnumFindFileList;
	fb_enum_find_file_entry			: FB_EnumFindFileEntry;
	fb_create_directory			: FB_CreateDir;	(* mit diesem FB kan nur eine Ordnerverzeichnissstruktur angelegt werden, jedoch keine Dateien erzeugt werden *)
	fb_file_open					: FB_FileOpen;	(* Eine vorhandene Datei öffnen oder eine Neue erzeugen *)
	fb_file_close					: FB_FileClose;
	fb_file_write					: FB_FileWrite;
	h_filehandle					: UINT := 0;(* file handle of the file *)
	arr_file_list					: ARRAY[0..63] OF ST_FindFileEntry;
	fb_ton_quitt					: TON;
	fb_r_trig_execute				: R_TRIG;
	fb_state_entry					: ST_StateEntry;
	temp_string					: STRING[255];
	i16_file_entry_zaehler			: INT := 0;
	i16_file_nr					: INT := 0;
	i							: INT := 0;
	b_pfad_vorhanden			: BOOL;
	b_datei_vorhanden			: BOOL;
END_VAR
fb_r_trig_execute(CLK:= bExecute, Q=> );
fb_ton_quitt(IN:= , PT:= t#100ms, Q=> , ET=> );

(* ======================================Schrittkette======================================== *)
fb_state_entry(
	i16_next_step:= ,
	i16_pos:= 1,
	s_debugtext:= ,
	E=> ,
	X=> ,
	i16_step=> ,
	i16_last_step=> );

CASE fb_state_entry.i16_step OF
(*=======================================================*)
	0:(* INIT *)
		bBusy := FALSE;
		bError := FALSE;
		nErrId := 0;
		fb_create_directory.bExecute := FALSE;
		fb_enum_find_file_list.bExecute := FALSE;
		fb_enum_find_file_entry.bExecute := FALSE;
		fb_file_open.bExecute := FALSE;
		fb_file_close.bExecute := FALSE;
		fb_state_entry.i16_next_step := 10;

(*=======================================================*)
	10:	(* Warte auf Execute-Befehl *)
		IF fb_state_entry.E THEN
			bBusy := FALSE;
		END_IF

		IF fb_r_trig_execute.Q THEN
			bBusy := TRUE;
			b_pfad_vorhanden := FALSE;
			b_datei_vorhanden := FALSE;
			fb_state_entry.i16_next_step := 20;
		END_IF

(*=======================================================*)
	20:	(* Prüfe, ob gewünschter Pfad auf dem Maschinen-PC vorhanden ist *)
		IF fb_state_entry.E THEN
			fb_enum_find_file_list.sPathName := s_path;
			fb_enum_find_file_list.eCmd := eEnumCmd_First;
			fb_enum_find_file_list.bExecute := TRUE;
		END_IF

		IF fb_enum_find_file_list.bBusy THEN
			fb_enum_find_file_list.bExecute := FALSE;
			fb_state_entry.i16_next_step := 30;
		END_IF

(*=======================================================*)
	30:	(* Auswerten des Ordner-Suchergebnis *)
		IF NOT fb_enum_find_file_list.bBusy THEN
			fb_enum_find_file_list.bExecute := FALSE;
		 	IF fb_enum_find_file_list.bError OR fb_enum_find_file_list.bEOE THEN
				 IF fb_enum_find_file_list.nFindFiles=0 THEN
					b_pfad_vorhanden := FALSE;
					fb_state_entry.i16_next_step := 40;	(* Pfad nicht vorhanden -> wird angelegt *)
				ELSE
					b_pfad_vorhanden := TRUE;
					fb_state_entry.i16_next_step := 60;	(* O.K. Pfad vorhanden -> Datei prüfen *)
				END_IF
			END_IF
		END_IF

(*=======================================================*)
	40:	(* Erstellen eines Ordnerverzeichnisses auf dem Laufwerk des Maschinen-PCs *)
		IF fb_state_entry.E THEN
			fb_create_directory.sPathName := s_path;
			fb_create_directory.bExecute := TRUE;
		END_IF

		IF fb_create_directory.bBusy THEN
			fb_create_directory.bExecute := FALSE;
			fb_state_entry.i16_next_step := 50;
		END_IF

(*=======================================================*)
	50:	(* Ordner wurde erstellt *)
		IF NOT fb_create_directory.bBusy  THEN
			IF NOT fb_create_directory.bError THEN
				fb_state_entry.i16_next_step := 60;	(* Ordnerverzeichnis wurde erfolgreich erstellt -> eine neue Datei anlegen oder eine Vorhandene öffnen *)
			ELSE
				fb_state_entry.i16_next_step := 1000;	(* Fehler *)
			END_IF
		END_IF

(*=======================================================*)
	60:	(* Prüfe, ob die gewünschte Datei in diesem Ordnerverzeichnis vorhanden ist *)
		IF fb_state_entry.E THEN
			temp_string := '';
			temp_string := CONCAT(temp_string, s_path);
			temp_string := CONCAT(temp_string, '\');
			temp_string := CONCAT(temp_string, s_dateiname);
			temp_string := CONCAT(temp_string, s_datei_erweiterung);
			fb_enum_find_file_entry.sPathName := temp_string;
			fb_enum_find_file_entry.eCmd := eEnumCmd_First;
			fb_enum_find_file_entry.bExecute := TRUE;
		END_IF

		IF fb_enum_find_file_entry.bBusy THEN
			fb_enum_find_file_entry.bExecute := FALSE;
			fb_state_entry.i16_next_step := 70;
		END_IF

(*=======================================================*)
	70:	(* Auswerten des Datei-Suchergebnis *)
		IF NOT fb_enum_find_file_entry.bBusy THEN
			fb_enum_find_file_entry.bExecute := FALSE;
		 	IF NOT fb_enum_find_file_entry.bError THEN
				IF fb_enum_find_file_entry.bEOE THEN
					IF fb_enum_find_file_entry.stFindFile.sFileName = CONCAT(s_dateiname, s_datei_erweiterung) THEN
					(* Datei bereits vorhanden *)
						b_datei_vorhanden := TRUE;
						fb_state_entry.i16_next_step := 0;
					ELSE
					(* Ende der Fileliste wurde erreicht und die gesuchte Datei ist  nicht vorhanden -> muss später angelegt werden *)
						b_datei_vorhanden := FALSE;
						fb_state_entry.i16_next_step := 100;
					END_IF
				ELSE
				(* Dateisuche im FB mit Abort korrekt beenden *)
					IF fb_enum_find_file_entry.stFindFile.sFileName = CONCAT(s_dateiname, s_datei_erweiterung) THEN
					(* Die gesuchte Datei wurde in der Fileliste gefunden *)
						b_datei_vorhanden := TRUE;
						fb_state_entry.i16_next_step := 80;
					ELSE
					(* Datei ist  nicht vorhanden -> muss später angelegt werden *)
						b_datei_vorhanden := FALSE;
						fb_state_entry.i16_next_step := 80;
					END_IF
				END_IF
			ELSE
				fb_state_entry.i16_next_step := FEHLER;
			END_IF
		END_IF

(*=======================================================*)
	80:	(* Dateisuchen wird beendet *)
		IF fb_state_entry.E THEN
			fb_enum_find_file_entry.eCmd := eEnumCmd_Abort;
			fb_enum_find_file_entry.bExecute := TRUE;
		END_IF

		IF fb_enum_find_file_entry.bBusy THEN
			fb_enum_find_file_entry.bExecute := FALSE;
			fb_state_entry.i16_next_step := 90;
		END_IF

(*=======================================================*)
	90:	(* Filehandle wieder frei *)
		IF NOT fb_enum_find_file_entry.bBusy THEN
			fb_enum_find_file_entry.bExecute := FALSE;
		 	IF NOT fb_enum_find_file_entry.bError AND fb_enum_find_file_entry.bEOE THEN
				fb_state_entry.i16_next_step := 100;
			ELSE
				fb_state_entry.i16_next_step := FEHLER;
			END_IF
		END_IF

(*=======================================================*)
	100:	(* Abfrage auf Datei anlegen *)
		IF fb_state_entry.E THEN
			IF NOT b_datei_vorhanden THEN
				fb_state_entry.i16_next_step := 110;
			ELSE
				fb_state_entry.i16_next_step := 0;	(* Fertig *)
			END_IF
		END_IF

(*=======================================================*)
	110:	(* Erzeugen einer neuen Datei *)
		IF fb_state_entry.E THEN
			temp_string := '';
			temp_string := CONCAT(temp_string, s_path);
			temp_string := CONCAT(temp_string, '\');
			temp_string := CONCAT(temp_string, s_dateiname);
			temp_string := CONCAT(temp_string, s_datei_erweiterung);
			fb_file_open.sPathName := temp_string;
			fb_file_open.nMode := FOPEN_MODEWRITE OR FOPEN_MODEBINARY;
			fb_file_open.bExecute := TRUE;
		END_IF

		IF fb_file_open.bBusy THEN
			fb_file_open.bExecute := FALSE;
			fb_state_entry.i16_next_step := 120;
		END_IF

(*=======================================================*)
	120:	(* Warte bis Datei geöffnet wurde *)
		IF NOT fb_file_open.bBusy  THEN
			IF NOT fb_file_open.bError THEN
				h_filehandle := fb_file_open.hFile;
				fb_state_entry.i16_next_step := 130;
			ELSE	(* Fehler *)
				nErrId := fb_file_open.nErrId;
				fb_state_entry.i16_next_step := 1000;
			END_IF
		END_IF

(*=======================================================*)
	130:	(* Schreibe die Dateistruktur im XML-Format: z.B.*)
		(*
		<Maschine1700_Datensicherung>
		<gst_datensatz>
		</gst_datensatz>
		</Maschine1700_Datensicherung>
		*)
		IF fb_state_entry.E THEN
			temp_string := '';
			temp_string := CONCAT(temp_string, '<');
			temp_string := CONCAT(temp_string, s_x_path_name);
			temp_string := CONCAT(temp_string, '>');
			temp_string := CONCAT(temp_string, '$r$n');

			(* Die Variable "s_xml_variablenname" wird hier schon mit angelegt, *)
			(* damit später beim "WECHSELN>" daraus gelesen werden kann, obwohl noch nichts drin steht *)
			temp_string := CONCAT(temp_string, '<');
			temp_string := CONCAT(temp_string, s_symname);
			temp_string := CONCAT(temp_string, '>');
			temp_string := CONCAT(temp_string, '$r$n');
			temp_string := CONCAT(temp_string, '<');
			temp_string := CONCAT(temp_string, '/');
			temp_string := CONCAT(temp_string, s_symname);
			temp_string := CONCAT(temp_string, '>');
			temp_string := CONCAT(temp_string, '$r$n');

			temp_string := CONCAT(temp_string, '<');
			temp_string := CONCAT(temp_string, '/');
			temp_string := CONCAT(temp_string, s_x_path_name);
			temp_string := CONCAT(temp_string, '>');
			fb_file_write.hFile := h_filehandle;
 			fb_file_write.bExecute := TRUE;
		END_IF

		IF fb_file_write.bBusy THEN
			fb_file_write.bExecute := FALSE;
			fb_state_entry.i16_next_step := 140;
		END_IF

(*=======================================================*)
	140:	(* Warte bis Datei geschrieben wurde *)
		IF NOT fb_file_write.bBusy  THEN
			IF NOT fb_file_write.bError THEN
				fb_state_entry.i16_next_step := 150;
			ELSE	(* Fehler *)
				nErrId := fb_file_write.nErrId;
				fb_state_entry.i16_next_step := 1000;
			END_IF
		END_IF

(*=======================================================*)
	150:	(* Schliesse Datei wieder, damit ein erneuter Zugriff möglich ist *)
		IF fb_state_entry.E THEN
			fb_file_close.hFile := h_filehandle;
			fb_file_close.bExecute := TRUE;
		END_IF

		IF fb_file_close.bBusy THEN
			fb_file_close.bExecute := FALSE;
			fb_state_entry.i16_next_step := 160;
		END_IF

(*=======================================================*)
	160:	(* Warte bis geschlossen *)
		IF NOT fb_file_close.bBusy  THEN
			IF NOT fb_file_close.bError THEN
				h_filehandle := 0;
				fb_state_entry.i16_next_step :=0;
			ELSE	(* Fehler *)
				nErrId := fb_file_close.nErrId;
				fb_state_entry.i16_next_step := 1000;
			END_IF
		END_IF

(*=======================================================*)
	1000: (* Fehler *)
		IF fb_state_entry.E THEN
			bBusy := FALSE;
			bError := TRUE;
			fb_ton_quitt.IN := FALSE;
		END_IF

		(*-----------------------Weiterschaltbedingungen----------------------------*)
		IF bQuit AND NOT fb_state_entry.E THEN
			bError := FALSE;
			fb_ton_quitt.IN := TRUE;
		END_IF

		IF fb_ton_quitt.Q THEN
			fb_ton_quitt.IN := FALSE;
			fb_state_entry.i16_next_step := 0;
		END_IF
END_CASE

fb_state_entry(
	i16_next_step:= , 
	i16_pos:= 2,
	s_debugtext:= ,
	E=> , 
	X=> , 
	i16_step=> ,
	i16_last_step=> );

fb_enum_find_file_list(
	sNetId:= '',
	sPathName:= ,
	eCmd:= ,
	pFindList:= ADR(arr_file_list),
	cbFindList:= SIZEOF(arr_file_list),
	bExecute:= ,
	tTimeout:= DEFAULT_ADS_TIMEOUT,
	bBusy=> ,
	bError=> ,
	nErrID=> , 
	bEOE=> ,
	nFindFiles=> );

fb_enum_find_file_entry(
	sNetId:= '',
	sPathName:= , 
	eCmd:= , 
	bExecute:= , 
	tTimeout:= DEFAULT_ADS_TIMEOUT,
	bBusy=> , 
	bError=> ,
	nErrID=> , 
	bEOE=> , 
	stFindFile=> );

fb_create_directory(
	sNetId:= '',
	sPathName:= ,
	ePath:= PATH_GENERIC,
	bExecute:= ,
	tTimeout:= DEFAULT_ADS_TIMEOUT,
	bBusy=> , 
	bError=> ,
	nErrId=> );

fb_file_open(
	sNetId:= '',
	sPathName:= , 
	nMode:= ,
	ePath:= PATH_GENERIC,
	bExecute:= , 
	tTimeout:= DEFAULT_ADS_TIMEOUT,
	bBusy=> , 
	bError=> , 
	nErrId=> , 
	hFile=> );

fb_file_close(
	sNetId:= '',
	hFile:= , 
	bExecute:= , 
	tTimeout:= t#10s,
	bBusy=> ,
	bError=> ,
	nErrId=> );

fb_file_write(
	sNetId:= '',
	hFile:= , 
	pWriteBuff:= ADR(temp_string),
	cbWriteLen:= LEN(temp_string),
	bExecute:= , 
	tTimeout:= t#10s,
	bBusy=> ,
	bError=> , 
	nErrId=> , 
	cbWrite=> );
END_FUNCTION_BLOCK

(* POU EPT Lib/Ethercat Diagnose/FB_EtherCatDiag, ST *)
FUNCTION_BLOCK FB_EtherCatDiag
VAR_INPUT
	st_config					: struct_config;
	st_ctrl_in					: struct_ctrl_in;
END_VAR
VAR_OUTPUT
	st_ctrl_out						: struct_ctrl_out;
END_VAR
VAR
	fb_state_entry					: ST_StateEntry;
	visu_Data						: struct_EthercatDiagnose;
	fb_ton_start						: TON;
	fb_ton_quitt						: TON;
	FB_EcGetAllSlaveStates			: FB_EcGetAllSlaveStates;
	by_AmsNetId					AT %I* : T_AmsNetIdArr;			(*Muss verknüpft werden*)
	s_AmsNetId					: T_AmsNetId := '0.0.0.0.0.0';	(* Master ID*)
	st_EcSlaveStateData			: ARRAY[1..MaxNoOfSlaves] OF ST_EcSlaveState;
	i_Slaves						: INT; 						(* Anzahl konfigurierter Slaves*)
	i								: INT;
	nErrId							: UDINT;

	sm_FehlerEthercat				: BOOL;

	FB_EcGetConfSlaves			: FB_EcGetConfSlaves;
	st_EcGetConfSlavesData		: ARRAY[1..MaxNoOfSlaves] OF ST_EcSlaveConfigData;


	fb_EcMasterFrameStatistic		: FB_EcMasterFrameStatistic;
END_VAR
(*======================================================
   ST: Fb_EtherCatDiag
 ------------------------------------------------------
   Auth: 	Thomas Vilgis, Werner Friedl    						 
   Date: 	25.01.2019    						     
   Rev.: 		1.1	
   Desc:		1.0	
				Der Baustein liest alle Zustände der Slaves aus.
   				Es muss nur die Variable "by_AmsNetId" mit dem EtherCAT Master verknüpt werden.
				Die maximale Anzahl an Slaves wird durch die globale Konstante "MaxNoOfSlaves" begrenzt.
				In der Visu werden die ausgelesenen Daten wie im Systemmanager angezeigt.
				Es wird eine Fehlermeldung ausgegeben, dass mindestens ein Teilnehmer nicht OP ist.
				Dies wird aber nur gemacht, wenn "st_config.b_station_aktiv" TRUE ist.
			1.1 
				UP und Down Button entfernt
				Var visu_Data.st_Slave[1].b_Err hinzugefüt => damit werden in der Visu Zeilen im Fehler farbig dargestellt.
			
   Historie: 	1.0

 ========================================================*)

(* Zeiten *)
fb_ton_start(IN:= NOT fb_ton_start.Q, PT:= T#2s, Q=>  , ET=> );
fb_ton_quitt(IN:= , PT:= t#100ms, Q=> , ET=> );
(* Flanken *)

(* ======================================Schrittkette======================================== *)
fb_state_entry(i16_pos:= 1);

CASE fb_state_entry.i16_step OF
(*=======================================================*)
	INIT_OBJ:	(*initialisieren*)

		(*-----------------------Weiterschaltbedingungen----------------------------*)
		IF st_config.b_config_fertig THEN
			fb_state_entry.i16_next_step:=INIT;
		END_IF
		
(*=======================================================*)
	INIT:	(*initialisieren*)
		IF fb_state_entry.E THEN
			fb_EcGetAllSlaveStates.bExecute := FALSE;
			fb_EcGetConfSlaves.bExecute := FALSE;
			fb_EcMasterFrameStatistic.bExecute := FALSE;
			sm_FehlerEthercat := FALSE;

			(*Umwandeln in einen String*)
			s_AmsNetId := F_CreateAmsNetId(by_AmsNetId);
		END_IF

		(*-----------------------Weiterschaltbedingungen----------------------------*)
		IF s_AmsNetId <> '0.0.0.0.0.0' THEN
			fb_state_entry.i16_next_step:=20;
		END_IF

(*=======================================================*)
	20:(* Baustein zum Abfragen der Configuration starten*)
		IF fb_state_entry.E THEN
			fb_EcGetConfSlaves.bExecute:=TRUE;
		END_IF

		(*-----------------------Weiterschaltbedingungen----------------------------*)
		IF 	fb_EcGetConfSlaves.bBusy THEN
			fb_state_entry.i16_next_step:=30;
		END_IF

(*=======================================================*)
	30:(* Warte auf Baustein *)

		(*-----------------------Weiterschaltbedingungen----------------------------*)
		IF NOT fb_EcGetConfSlaves.bBusy THEN
			fb_EcGetConfSlaves.bExecute:=FALSE;
			IF 	fb_EcGetConfSlaves.bError THEN
				nErrId:=fb_EcGetConfSlaves.nErrorId;
				fb_state_entry.i16_next_step:=FEHLER;
			ELSE
				fb_state_entry.i16_next_step:=BEREIT;
			END_IF
		END_IF
		
(*=======================================================*)
	BEREIT:	(*  *)
		IF fb_state_entry.E THEN
			LeseDaten();
		END_IF

		(*-----------------------Weiterschaltbedingungen----------------------------*)
		IF fb_ton_start.Q THEN
			fb_state_entry.i16_next_step:=110;
		END_IF

(*=======================================================*)
	110:(* Baustein zum Abfragen des Status starten*)
		IF fb_state_entry.E THEN
			fb_EcGetAllSlaveStates.bExecute:=TRUE;
		END_IF

		(*-----------------------Weiterschaltbedingungen----------------------------*)
		IF 	fb_EcGetAllSlaveStates.bBusy THEN
			fb_state_entry.i16_next_step:=120;
		END_IF

(*=======================================================*)
	120:(* Warte auf Baustein *)

		(*-----------------------Weiterschaltbedingungen----------------------------*)
		IF NOT fb_EcGetAllSlaveStates.bBusy THEN
			fb_EcGetAllSlaveStates.bExecute:=FALSE;
			IF 	fb_EcGetAllSlaveStates.bError THEN
				nErrId:=fb_EcGetAllSlaveStates.nErrId;
				fb_state_entry.i16_next_step:=FEHLER;
			ELSE
				i_Slaves := UINT_TO_INT(fb_EcGetAllSlaveStates.nSlaves);
				fb_state_entry.i16_next_step:=130;
			END_IF
		END_IF

(*=======================================================*)
	130:(* Prüfe, ob ein Slave einen Fehler hat *)
		IF fb_state_entry.E THEN
			sm_FehlerEthercat := FALSE;
			(*Fehlermeldung nur ausgeben, wenn Sation aktiv ist*)
			IF st_config.b_station_aktiv THEN
				FOR i:= 1 TO i_Slaves DO
					IF st_EcSlaveStateData[i].deviceState <> EC_DEVICE_STATE_OP THEN
						visu_Data.st_Slave[i].b_Err:=TRUE;
						sm_FehlerEthercat := TRUE;
						(*-----------------------Weiterschaltbedingungen----------------------------*)
						fb_state_entry.i16_next_step:=FEHLER;
					ELSE
						visu_Data.st_Slave[i].b_Err:=FALSE;
						(*-----------------------Weiterschaltbedingungen----------------------------*)
						fb_state_entry.i16_next_step:=140;
					END_IF
				END_FOR
			END_IF
		END_IF

(*=======================================================*)
	140:(* Baustein zum Abfragen der Lost Frames starten*)
		IF fb_state_entry.E THEN
			fb_EcMasterFrameStatistic.bExecute:=TRUE;
		END_IF

		(*-----------------------Weiterschaltbedingungen----------------------------*)
		IF 	fb_EcMasterFrameStatistic.bBusy THEN
			fb_state_entry.i16_next_step:=150;
		END_IF

(*=======================================================*)
	150:(* Warte auf Baustein *)

		(*-----------------------Weiterschaltbedingungen----------------------------*)
		IF NOT fb_EcMasterFrameStatistic.bBusy THEN
			fb_EcMasterFrameStatistic.bExecute:=FALSE;
			IF 	fb_EcMasterFrameStatistic.bError THEN
				nErrId:=fb_EcMasterFrameStatistic.nErrId;
				fb_state_entry.i16_next_step:=FEHLER;
			ELSE
				fb_state_entry.i16_next_step:=BEREIT;
			END_IF
		END_IF



(*=======================================================*)
	FEHLER:
		IF fb_state_entry.E THEN
			fb_ton_quitt.IN := FALSE;
			st_ctrl_out.b_fehler := TRUE;
		END_IF

		(*-----------------------Weiterschaltbedingungen----------------------------*)
		IF st_ctrl_in.b_quitt AND NOT fb_state_entry.E THEN
			st_ctrl_out.b_fehler := FALSE;
			fb_ton_quitt.IN := TRUE;
		END_IF

		IF fb_ton_quitt.Q THEN
			fb_ton_quitt.IN := FALSE;
			fb_state_entry.i16_next_step := INIT;
		END_IF

END_CASE


fb_state_entry(i16_pos:= 2);


(*Aufruf*)
fb_EcGetAllSlaveStates(
	sNetId:= s_AmsNetId, 
	pStateBuf:= ADR(st_EcSlaveStateData),
	cbBufLen:= SIZEOF(st_EcSlaveStateData));

fb_EcGetConfSlaves(
	sNetId:= s_AmsNetId,
	pArrEcConfSlaveInfo:= ADR(st_EcGetConfSlavesData),
	cbBufLen:= SIZEOF(st_EcGetConfSlavesData) );

fb_EcMasterFrameStatistic(
	sNetId:= s_AmsNetId);
	


IF st_config.b_config_fertig THEN
	(* Fehlermeldungen und Betriebsmeldungen ab dem Startindex in die globalen Meldungsarrays schreiben *)
	garr_stoermeldungen[st_config.i16_meld_startindex + 0] := sm_FehlerEthercat;
	garr_stoermeldungen[st_config.i16_meld_startindex + 1] := FALSE;
	garr_stoermeldungen[st_config.i16_meld_startindex + 2] := FALSE;
	garr_stoermeldungen[st_config.i16_meld_startindex + 3] := FALSE;
	garr_stoermeldungen[st_config.i16_meld_startindex + 4] := FALSE;

	garr_betriebsmeldungen[st_config.i16_meld_startindex + 0] := FALSE;
	garr_betriebsmeldungen[st_config.i16_meld_startindex + 1] := FALSE;
	garr_betriebsmeldungen[st_config.i16_meld_startindex + 2] := FALSE;
	garr_betriebsmeldungen[st_config.i16_meld_startindex + 3] := FALSE;
	garr_betriebsmeldungen[st_config.i16_meld_startindex + 4] := FALSE;
END_IF
END_FUNCTION_BLOCK
ACTION LeseDaten:
(*Master Daten übergeben*)
visu_Data.ST_Master.s_Name := st_config.str_instanz_name;
visu_Data.st_Master.s_AmsNetId := s_AmsNetId;
visu_Data.st_Master.i_Slaves := i_Slaves;
visu_Data.st_Master.f_FramesPerSeconed := fb_EcMasterFrameStatistic.fFramesPerSecond;
visu_Data.st_Master.i_LostFrames := fb_EcMasterFrameStatistic.nLostFrames;

(*Slave Daten übergeben*)
FOR i:=1 TO MaxNoOfSlaves DO
	visu_Data.st_Slave[i].i_Number := i;
	IF st_EcGetConfSlavesData[i].nAddr <> 0 THEN
		visu_Data.st_Slave[i].s_Adress := WORD_TO_STRING(st_EcGetConfSlavesData[i].nAddr);
	END_IF
	visu_Data.st_Slave[i].s_Name := st_EcGetConfSlavesData[i].sName;
	visu_Data.st_Slave[i].s_Type := st_EcGetConfSlavesData[i].sType;

	visu_Data.st_Slave[i].s_DeviceState := F_ConvStateToString(st_EcSlaveStateData[i].deviceState);

	(*Link State wird von TwinCAT aus Status und Port-Nummer zusammengebaut*)
	CASE st_EcSlaveStateData[i].linkState OF
		0:
			;	(*alles OK*)
		1:
			visu_Data.st_Slave[i].s_DeviceState := CONCAT(visu_Data.st_Slave[i].s_DeviceState, ' NO_COMM');
			
		18:
			visu_Data.st_Slave[i].s_DeviceState := CONCAT(visu_Data.st_Slave[i].s_DeviceState, ' LINK_WITHOUT_COMM A');
		34:
			visu_Data.st_Slave[i].s_DeviceState := CONCAT(visu_Data.st_Slave[i].s_DeviceState, ' LINK_WITHOUT_COMM B');
		66:
			visu_Data.st_Slave[i].s_DeviceState := CONCAT(visu_Data.st_Slave[i].s_DeviceState, ' LINK_WITHOUT_COMM C');
		130:
			visu_Data.st_Slave[i].s_DeviceState := CONCAT(visu_Data.st_Slave[i].s_DeviceState, ' LINK_WITHOUT_COMM D');
			
		20:
			visu_Data.st_Slave[i].s_DeviceState := CONCAT(visu_Data.st_Slave[i].s_DeviceState, ' MISSING_LINK A');
		36:
			visu_Data.st_Slave[i].s_DeviceState := CONCAT(visu_Data.st_Slave[i].s_DeviceState, ' MISSING_LINK B');
		68:
			visu_Data.st_Slave[i].s_DeviceState := CONCAT(visu_Data.st_Slave[i].s_DeviceState, ' MISSING_LINK C');
		132:
			visu_Data.st_Slave[i].s_DeviceState := CONCAT(visu_Data.st_Slave[i].s_DeviceState, ' MISSING_LINK D');
			
		24:
			visu_Data.st_Slave[i].s_DeviceState := CONCAT(visu_Data.st_Slave[i].s_DeviceState, ' ADDITIONAL_LINK A');
		40:
			visu_Data.st_Slave[i].s_DeviceState := CONCAT(visu_Data.st_Slave[i].s_DeviceState, ' ADDITIONAL_LINK B');
		72:
			visu_Data.st_Slave[i].s_DeviceState := CONCAT(visu_Data.st_Slave[i].s_DeviceState, ' ADDITIONAL_LINK C');
		136:
			visu_Data.st_Slave[i].s_DeviceState := CONCAT(visu_Data.st_Slave[i].s_DeviceState, ' ADDITIONAL_LINK D');
		
		ELSE
			visu_Data.st_Slave[i].s_DeviceState := CONCAT(visu_Data.st_Slave[i].s_DeviceState, ' undefined');
	END_CASE
END_FOR
END_ACTION

(* POU Gemeinsamkeiten17xx/XML Server/FB_XMLFileCopy, ST *)
FUNCTION_BLOCK FB_XMLFileCopy
VAR_INPUT
	srcNetId				: T_AmsNetId;	(* TwinCAT network address of the source file *)
	destNetId			: T_AmsNetId;	(* TwinCAT network address of the destination file *)
	bExecute			: BOOL;
	bQuit				: BOOL;
	s_name_quelldatei	: STRING;
	s_name_zieldatei		: STRING;
END_VAR
VAR_OUTPUT
	bBusy				: BOOL;
	bError				: BOOL;
	nErrId				: UDINT;
END_VAR
VAR
	fb_file_open			: FB_FileOpen;
	fb_file_close			: FB_FileClose;
	fb_file_read			: FB_FileRead;
	fb_file_write			: FB_FileWrite;

	h_quell_filehandle		: UINT := 0;(* file handle of the source file *)
	h_ziel_filehandle		: UINT := 0;(* file handle of the destination file *)

	fb_state_entry			: ST_StateEntry;
	fb_r_trig_execute		: R_TRIG;
	fb_ton_quitt			: TON;
	p_read_write_buffer	: ARRAY[1..100000] OF BYTE;
	cb_write_length		: UDINT :=0;
	cb_read_length		: UDINT :=0;
END_VAR
fb_r_trig_execute(CLK:= bExecute, Q=> );
fb_ton_quitt(IN:= , PT:= t#100ms, Q=> , ET=> );

(* ======================================Schrittkette======================================== *)
fb_state_entry(
	i16_next_step:= ,
	i16_pos:= 1,
	s_debugtext:= ,
	E=> ,
	X=> ,
	i16_step=> ,
	i16_last_step=> );

CASE fb_state_entry.i16_step OF
(*=======================================================*)
	0:(* INIT *)
		bBusy := FALSE;
		bError := FALSE;
		nErrId := 0;
		fb_file_open.bExecute := FALSE;
		fb_file_close.bExecute := FALSE;
		fb_file_read.bExecute := FALSE;
		fb_file_write.bExecute := FALSE;
		h_quell_filehandle := 0;
		h_ziel_filehandle := 0;
		cb_write_length :=0;
		cb_read_length :=0;
		fb_state_entry.i16_next_step := 10;

(*=======================================================*)
	10:	(* Warte auf Execute-Befehl *)
		IF fb_state_entry.E THEN
			bBusy := FALSE;
		END_IF

		IF fb_r_trig_execute.Q THEN
			bBusy := TRUE;
			fb_state_entry.i16_next_step := 100;
		END_IF

(*=======================================================*)
	100:	(* Öffne Quelldatei *)
		IF fb_state_entry.E THEN
			fb_file_open.nMode := FOPEN_MODEREAD OR FOPEN_MODEBINARY;
			fb_file_open.sPathName := s_name_quelldatei;
			fb_file_open.bExecute := TRUE;
		END_IF

		IF fb_file_open.bBusy THEN
			fb_file_open.bExecute := FALSE;
			fb_state_entry.i16_next_step := 110;
		END_IF

(*=======================================================*)
	110:	(* Warte bis Quelle geöffnet *)
		IF NOT fb_file_open.bBusy  THEN
			IF NOT fb_file_open.bError THEN
				h_quell_filehandle := fb_file_open.hFile;
				fb_state_entry.i16_next_step := 120;
			ELSE	(* Fehler *)
				nErrId := fb_file_open.nErrId;
				fb_state_entry.i16_next_step := 300;
			END_IF
		END_IF

(*=======================================================*)
	120:	(* Öffne Zieldatei *)
		IF fb_state_entry.E THEN
			fb_file_open.nMode := FOPEN_MODEWRITE OR FOPEN_MODEBINARY;
			fb_file_open.sPathName := s_name_zieldatei;
			fb_file_open.bExecute := TRUE;
		END_IF

		IF fb_file_open.bBusy THEN
			fb_file_open.bExecute := FALSE;
			fb_state_entry.i16_next_step := 130;
		END_IF

(*=======================================================*)
	130:	(* Warte bis Ziel geöffnet *)
		IF NOT fb_file_open.bBusy  THEN
			IF NOT fb_file_open.bError THEN
				h_ziel_filehandle := fb_file_open.hFile;
				fb_state_entry.i16_next_step := 150;
			ELSE	(* Fehler *)
				nErrId := fb_file_open.nErrId;
				fb_state_entry.i16_next_step := 300;
			END_IF
		END_IF

(*=======================================================*)
	150:	(* Lese Daten von der Quelldatei *)
		IF fb_state_entry.E THEN
			fb_file_read.hFile := h_quell_filehandle;
			fb_file_read.bExecute := TRUE;
		END_IF

		IF fb_file_read.bBusy THEN
			fb_file_read.bExecute := FALSE;
			fb_state_entry.i16_next_step := 160;
		END_IF

(*=======================================================*)
	160:	(* Warte bis gelesen *)
		IF NOT fb_file_read.bBusy  THEN
			IF NOT fb_file_read.bError THEN
				cb_read_length := fb_file_read.cbRead;
				fb_state_entry.i16_next_step := 170;
			ELSE	(* Fehler *)
				nErrId := fb_file_read.nErrId;
				fb_state_entry.i16_next_step := 300;
			END_IF
		END_IF

(*=======================================================*)
	170:	(* Schreibe Daten in die Zieldatei *)
		IF fb_state_entry.E THEN
			fb_file_write.hFile := h_ziel_filehandle;
			cb_write_length := cb_read_length;
			fb_file_write.bExecute := TRUE;
		END_IF

		IF fb_file_write.bBusy THEN
			fb_file_write.bExecute := FALSE;
			fb_state_entry.i16_next_step := 180;
		END_IF

(*=======================================================*)
	180:	(* Warte bis geschrieben *)
		IF NOT fb_file_write.bBusy  THEN
			IF NOT fb_file_write.bError THEN
				IF fb_file_read.bEOF THEN (* Prüfe, ob das EOF-Flag gesetzt ist *)
					fb_state_entry.i16_next_step := 200; (* Quell- und Zieldatei schliessen *)
				ELSE
					fb_state_entry.i16_next_step := 150; (* Weitere Daten lesen *)
				END_IF
			ELSE	(* Fehler *)
				nErrId := fb_file_write.nErrId;
				fb_state_entry.i16_next_step := 300;
			END_IF
		END_IF

(*=======================================================*)
	200:	(* Schliessen der Zieldatei *)
		IF fb_state_entry.E THEN
			fb_file_close.hFile := h_ziel_filehandle;
			fb_file_close.bExecute := TRUE;
		END_IF

		IF fb_file_close.bBusy THEN
			fb_file_close.bExecute := FALSE;
			fb_state_entry.i16_next_step := 210;
		END_IF

(*=======================================================*)
	210:	(* Warte bis Ziel geschlossen *)
		IF NOT fb_file_close.bBusy  THEN
			IF NOT fb_file_close.bError THEN
				h_ziel_filehandle := 0;
				fb_state_entry.i16_next_step := 220;
			ELSE	(* Fehler *)
				nErrId := fb_file_close.nErrId;
				fb_state_entry.i16_next_step := 300;
			END_IF
		END_IF

(*=======================================================*)
	220:	(* Schliessen der Quelldatei *)
		IF fb_state_entry.E THEN
			fb_file_close.hFile := h_quell_filehandle;
			fb_file_close.bExecute := TRUE;
		END_IF

		IF fb_file_close.bBusy THEN
			fb_file_close.bExecute := FALSE;
			fb_state_entry.i16_next_step := 230;
		END_IF

(*=======================================================*)
	230:	(* Warte bis Quelle geschlossen *)
		IF NOT fb_file_close.bBusy  THEN
			IF NOT fb_file_close.bError THEN
				h_quell_filehandle := 0;
				fb_state_entry.i16_next_step := 10;
			ELSE	(* Fehler *)
				nErrId := fb_file_close.nErrId;
				fb_state_entry.i16_next_step := 300;
			END_IF
		END_IF

(*=======================================================*)
	300:	(* Bei Fehler müssen Quell- und Zieldatei auf jeden Fall geschlossen werden *)
		(* Beide Dateien korrekt geschlossen -> Fehler auswerten *)
		IF ( h_ziel_filehandle = 0 AND h_quell_filehandle = 0 ) THEN
			fb_state_entry.i16_next_step := 1000;
		(* Beide Dateien sind noch offen und müsse zuerst geschlossen werden -> schliesse zuerst die Quelle*)
		ELSIF (h_quell_filehandle <> 0 AND h_ziel_filehandle <> 0 ) THEN
			fb_file_close.hFile := h_quell_filehandle;
			fb_state_entry.i16_next_step := 310;
		(* Quelle offen und Ziel geschlossen -> Quelle schliessen *)
		ELSIF (h_quell_filehandle <> 0 AND h_ziel_filehandle = 0 ) THEN
			fb_file_close.hFile := h_quell_filehandle;
			fb_state_entry.i16_next_step := 310; (* Schliesse Quelldatei *)
		(* Ziel offen und Quelle geschlossen -> Ziel schliessen *)
		ELSIF (h_quell_filehandle = 0 AND h_ziel_filehandle <> 0) THEN
			fb_file_close.hFile := h_ziel_filehandle;
			fb_state_entry.i16_next_step := 310; (* Schliesse Zielldatei *)
			bBusy := FALSE;
		END_IF

(*=======================================================*)
	310:	(* Schliessen der Datei *)
		IF fb_state_entry.E THEN
			fb_file_close.bExecute := TRUE;
		END_IF

		IF fb_file_close.bBusy THEN
			fb_file_close.bExecute := FALSE;
			fb_state_entry.i16_next_step := 320;
		END_IF

(*=======================================================*)
	320:	(* Warte bis geschlossen *)
		IF NOT fb_file_close.bBusy  THEN
			IF NOT fb_file_close.bError THEN
				IF fb_file_close.hFile = h_quell_filehandle THEN
					h_quell_filehandle := 0;
				ELSIF fb_file_close.hFile = h_ziel_filehandle THEN
					h_ziel_filehandle := 0;
				END_IF
				fb_state_entry.i16_next_step := 300;
			ELSE	(* Fehler *)
				nErrId := fb_file_close.nErrId;
				fb_state_entry.i16_next_step := 1000;
			END_IF
		END_IF

(*=======================================================*)
	1000: (* Fehler *)
		IF fb_state_entry.E THEN
			bBusy := FALSE;
			bError := TRUE;
			fb_ton_quitt.IN := FALSE;
		END_IF

		(*-----------------------Weiterschaltbedingungen----------------------------*)
		IF bQuit AND NOT fb_state_entry.E THEN
			bError := FALSE;
			fb_ton_quitt.IN := TRUE;
		END_IF

		IF fb_ton_quitt.Q THEN
			fb_ton_quitt.IN := FALSE;
			fb_state_entry.i16_next_step := 0;
		END_IF
END_CASE

fb_state_entry(
	i16_next_step:= , 
	i16_pos:= 2,
	s_debugtext:= ,
	E=> , 
	X=> , 
	i16_step=> ,
	i16_last_step=> );

fb_file_close(
	sNetId:= '',
	hFile:= , 
	bExecute:= , 
	tTimeout:= DEFAULT_ADS_TIMEOUT,
	bBusy=> ,
	bError=> , 
	nErrId=> );

fb_file_open(
	sNetId:= '',
	sPathName:= ,
	nMode:= 	,
	ePath:= PATH_GENERIC,
	bExecute:= , 
	tTimeout:= DEFAULT_ADS_TIMEOUT,
	bBusy=> ,
	bError=> , 
	nErrId=> ,
	hFile=> );

fb_file_read(
	sNetId:= ,
	hFile:= , 
	pReadBuff:= ADR(p_read_write_buffer),
	cbReadLen:= SIZEOF(p_read_write_buffer),
	bExecute:= , 
	tTimeout:= DEFAULT_ADS_TIMEOUT,
	bBusy=> , 
	bError=> ,
	nErrId=> ,
	cbRead=> , 
	bEOF=> );

fb_file_write(
	sNetId:= ,
	hFile:= ,
	pWriteBuff:= ADR(p_read_write_buffer),
	cbWriteLen:= cb_write_length,
	bExecute:= , 
	tTimeout:= DEFAULT_ADS_TIMEOUT,
	bBusy=> , 
	bError=> , 
	nErrId=> , 
	cbWrite=> );
END_FUNCTION_BLOCK

(* POU EPT Lib/Programmbausteine/Routing/ADS-Kommunikation/ReadAdsStruct, ST *)
FUNCTION_BLOCK ReadAdsStruct
VAR_INPUT
	b_Execute				: BOOL;
	b_Reset					: BOOL;
	AmsNetId				: STRING;
	Port						: UINT;
	s_SymbolName			: STRING;
	dw_DestAdr				: DWORD;
END_VAR
VAR_OUTPUT
	b_Busy					: BOOL;
	b_Done					: BOOL;
	b_Error					: BOOL;
	b_ErrorID				: UDINT;
END_VAR
VAR
	s_SymbolNameOld		: STRING;
	str_SymInfo				: SYMINFOSTRUCT;

	fb_read_symbolinfo		: PLC_ReadSymInfoByName;
	fb_ads_read				: ADSREAD;

	Done					: BOOL;
	fb_ton_quitt				: TON;
	fb_state_entry				: ST_StateEntry;
END_VAR
fb_ton_quitt(IN:= , PT:= t#1s, Q=> , ET=> );

fb_state_entry(
	i16_next_step:= , 
	i16_pos:= 1,
	s_debugtext:= ,
	E=> ,
	X=> ,
	i16_step=> ,
	i16_last_step=> );

CASE fb_state_entry.i16_step OF
(*=======================================================*)
	0:
		IF b_Execute THEN
			fb_state_entry.i16_next_step := 10;
		END_IF

(*=======================================================*)
	10:	(* Get Symbolinfo if necessary *)
		b_Busy := TRUE;
		IF str_SymInfo.idxGroup <> 0 AND s_SymbolName = s_SymbolNameOld THEN
			fb_state_entry.i16_next_step := 100;
		ELSE
			fb_state_entry.i16_next_step := 20;
		END_IF

(*=======================================================*)
	20:	(* Read Symbolinfo *)
		fb_read_symbolinfo.START := TRUE;
		IF fb_read_symbolinfo.BUSY THEN
			fb_state_entry.i16_next_step := 30;
		END_IF

(*=======================================================*)
	30:	(* Done or Error *)
		IF NOT fb_read_symbolinfo.BUSY THEN
			IF NOT fb_read_symbolinfo.ERR THEN
				fb_read_symbolinfo.START := FALSE;
				s_SymbolNameOld := s_SymbolName;
				fb_state_entry.i16_next_step := 100;
			ELSE
				b_Error := TRUE;
				b_ErrorID := fb_read_symbolinfo.ERRID;
				fb_state_entry.i16_next_step := 1000;
			END_IF
		END_IF

(*=======================================================*)
	100:	(* Read Symbol-Data *)
			fb_ads_read.READ := TRUE;
			IF fb_ads_read.BUSY THEN
				fb_state_entry.i16_next_step := 110;
			END_IF

(*=======================================================*)
	110:	(* Read is Busy *)
		IF NOT fb_ads_read.BUSY THEN
			IF NOT fb_ads_read.ERR THEN
				fb_ads_read.READ := FALSE;
				b_Done := TRUE;
				b_Busy := FALSE;
				fb_state_entry.i16_next_step := 120;
			ELSE
				b_Error := TRUE;
				b_ErrorID := fb_ads_read.ERRID;
				fb_state_entry.i16_next_step := 1000;
			END_IF
		END_IF

(*=======================================================*)
	120:	(* Read erfolgreich abgeschlossen *)
		IF NOT b_Execute THEN
			b_Done := FALSE;
			b_Busy := FALSE;
			fb_state_entry.i16_next_step := 0;
		END_IF;

(*=======================================================*)
	1000:	(* Fehler *)
		fb_read_symbolinfo.START := FALSE;
		fb_ads_read.READ := FALSE;

		IF b_Reset THEN
			fb_state_entry.i16_next_step := 0;
			b_Done := FALSE;
			b_Busy := FALSE;
			b_Error := FALSE;
			b_ErrorID := 0;
		END_IF

END_CASE

fb_state_entry(
	i16_next_step:= , 
	i16_pos:= 2,
	s_debugtext:= ,
	E=> , 
	X=> ,
	i16_step=> ,
	i16_last_step=> );

fb_read_symbolinfo(
	NETID:= AmsNetId,
	PORT:= Port,
	SYMNAME:= s_SymbolName,
	START:= , 
	TMOUT:= DEFAULT_ADS_TIMEOUT,
	BUSY=> , 
	ERR=> , 
	ERRID=> , 
	SYMINFO=> str_SymInfo);

fb_ads_read(
	NETID:= AmsNetId,
	PORT:= Port,
	IDXGRP:= str_SymInfo.idxGroup,
	IDXOFFS:= str_SymInfo.idxOffset,
	LEN:= str_SymInfo.byteSize,
	DESTADDR:= dw_DestAdr,
	READ:= , 
	TMOUT:= DEFAULT_ADS_TIMEOUT,
	BUSY=> , 
	ERR=> , 
	ERRID=> );
END_FUNCTION_BLOCK

(* POU EPT Lib/Funktionen/Scale, ST *)
FUNCTION Scale : REAL
VAR_INPUT
	i16Messwert : INT;
	i16MessbereichUnten : INT;
	i16MessbereichOben : INT;
	rSkaleUnten : REAL;
	rSkaleOben : REAL;
END_VAR
VAR
END_VAR
(* Überwachung auf Division durch Null*)
IF i16MessbereichOben <> i16MessbereichUnten THEN

Scale := ( rSkaleOben - rSkaleUnten ) * i16Messwert / ( i16MessbereichOben - i16MessbereichUnten );

END_IF
END_FUNCTION

(* POU EPT Lib/Programmbausteine/Routing/ADS-Kommunikation/ST_ADS_Kommunikation, ST *)
FUNCTION_BLOCK ST_ADS_Kommunikation
VAR_INPUT
	s_read_symbol_name			: STRING;
	s_write_symbol_name			: STRING;
	dw_read_source_adr_vorher	: struct_station_vorher_out;
	dw_write_source_adr_vorher	: struct_station_vorher_in;
	dw_read_source_adr_nachher	: struct_station_nachher_out;
	dw_write_source_adr_nachher	: struct_station_nachher_in;
END_VAR
VAR
	fb_read_ads					: ReadAdsStruct;
	fb_write_ads					: WriteAdsStruct;

	fb_ton_wz					: TON;
	fb_ton_quitt					: TON;
	fb_state_entry					: ST_StateEntry;
	b_ibn_start					: BOOL := FALSE;
	fb_r_trig_ibn_start				: R_TRIG;
	fb_ton_ibn_start				: TON;
	s_AMSNetId					: STRING;
END_VAR
(* Zeiten *)
fb_ton_wz(IN:= , PT:= , Q=> , ET=> );
fb_ton_quitt(IN:= , PT:= t#3s, Q=> , ET=> );

fb_r_trig_ibn_start(CLK:= b_ibn_start, Q=> );
fb_ton_ibn_start(IN:= , PT:= t#1s, Q=> , ET=> );

IF fb_r_trig_ibn_start.Q THEN
	fb_ton_ibn_start.IN := TRUE;
ELSE
	IF fb_ton_ibn_start.Q THEN
		b_ibn_start := FALSE;
	 	fb_ton_ibn_start.IN := FALSE;
	END_IF
END_IF

fb_state_entry(
	i16_next_step:= , 
	i16_pos:= 1,
	s_debugtext:= ,
	E=> ,
	X=> ,
	i16_step=> ,
	i16_last_step=> );

CASE fb_state_entry.i16_step OF
(*=======================================================*)
	0:	(* Initialisierung *)
		fb_read_ads.b_Execute := FALSE;
		fb_write_ads.b_Execute := FALSE;
		fb_read_ads.b_Reset := FALSE;
		fb_write_ads.b_Reset := FALSE;
		fb_ton_wz.IN := FALSE;
		fb_state_entry.i16_next_step := 10;

(*=======================================================*)
	10:	(* Warte bis Routing-Verbindung zum Front-PC wurde angelegt wurde *)
		IF fb_state_entry.E THEN
			;
		END_IF

		(*-----------------------Weiterschaltbedingungen----------------------------*)
		IF ST_RoutingBackpanel.fb_state_entry.i16_step = 999 THEN
			fb_state_entry.i16_next_step := 20;
		END_IF

(*=======================================================*)
	20:	(* Lese NetId von angeschlossenen Remote-PCs *)
		IF fb_state_entry.E THEN
			s_AMSNetId :=  ST_RoutingBackpanel.s_backpanel_netid;
		END_IF

		fb_state_entry.i16_next_step := 100;

(*==========================LESEN=============================*)
	100:	(* Lesen der Symbole über ADS *)
		IF fb_state_entry.E THEN
			fb_read_ads.b_Execute := TRUE;
		END_IF

		IF fb_read_ads.b_Busy THEN
			fb_read_ads.b_Execute := FALSE;
			fb_state_entry.i16_next_step := 110;
		END_IF

(*=======================================================*)
	110:	(* Lesen abgeschlossen *)
		IF NOT fb_read_ads.b_Busy AND fb_read_ads.b_Done THEN
			fb_state_entry.i16_next_step := 200;
		ELSIF fb_read_ads.b_Error THEN
			fb_state_entry.i16_next_step := 1000;
		END_IF

(*===========================SCHREIBEN============================*)
	200:	(* Schreiben der Symbole über ADS *)
		IF fb_state_entry.E THEN
			fb_write_ads.b_Execute := TRUE;
		END_IF

		IF fb_write_ads.b_Busy THEN
			fb_write_ads.b_Execute := FALSE;
			fb_state_entry.i16_next_step := 210;
		END_IF

(*=======================================================*)
	210:	(* Schreiben abgeschlossen *)
		IF NOT fb_write_ads.b_Busy AND fb_write_ads.b_Done THEN
			fb_state_entry.i16_next_step := 999;
		ELSIF fb_write_ads.b_Error THEN
			fb_state_entry.i16_next_step := 1000;
		END_IF

(*=======================================================*)
	999:	(* Ende *)
		fb_state_entry.i16_next_step := 100;

(*=======================================================*)
	1000:	(* Fehler *)
		IF fb_state_entry.E THEN
			fb_read_ads.b_Execute := FALSE;
			fb_write_ads.b_Execute := FALSE;
			fb_ton_wz.IN := FALSE;
			fb_ton_quitt.IN := TRUE;
		END_IF

		IF  fb_ton_quitt.Q THEN
			fb_ton_quitt.IN := FALSE;
			fb_read_ads.b_Reset := TRUE;
			fb_write_ads.b_Reset := TRUE;
			fb_state_entry.i16_next_step := 0;
		END_IF
END_CASE

fb_state_entry(
	i16_next_step:= , 
	i16_pos:= 2,
	s_debugtext:= ,
	E=> , 
	X=> ,
	i16_step=> ,
	i16_last_step=> );

fb_read_ads(
	b_Execute:= ,
	b_Reset:= ,
	AmsNetId:= s_AMSNetId ,
	Port:= 801,
	s_SymbolName:=s_read_symbol_name ,
	dw_DestAdr:= ADR(dw_read_source_adr_vorher),
	b_Busy=> ,
	b_Done=> ,
	b_Error=> ,
	b_ErrorID=> );

fb_write_ads(
	b_Execute:= ,
	b_Reset:= ,
	AmsNetId:= s_AMSNetId,
	Port:= 801 ,
	s_SymbolName:=  s_write_symbol_name,
	dw_SourceAdr:= ADR(dw_write_source_adr_vorher) ,
	b_Busy=> ,
	b_Done=> ,
	b_Error=> ,
	b_ErrorID=> );
END_FUNCTION_BLOCK

(* POU EPT Lib/Programmbausteine/Routing/ADS-Kommunikation/WriteAdsStruct, ST *)
FUNCTION_BLOCK WriteAdsStruct
VAR_INPUT
	b_Execute				: BOOL;
	b_Reset					: BOOL;
	AmsNetId				: STRING;
	Port						: UINT;
	s_SymbolName			: STRING;
	dw_SourceAdr			: DWORD;
END_VAR
VAR_OUTPUT
	b_Busy					: BOOL;
	b_Done					: BOOL;
	b_Error					: BOOL;
	b_ErrorID				: UDINT;
END_VAR
VAR
	s_SymbolNameOld		: STRING;
	str_SymInfo				: SYMINFOSTRUCT;

	fb_read_symbolinfo		: PLC_ReadSymInfoByName;
	fb_ads_write				: ADSWRITE;

	Done					: BOOL;
	fb_ton_quitt				: TON;
	fb_state_entry				: ST_StateEntry;
END_VAR
fb_ton_quitt(IN:= , PT:= t#1s, Q=> , ET=> );

fb_state_entry(
	i16_next_step:= , 
	i16_pos:= 1,
	s_debugtext:= ,
	E=> ,
	X=> ,
	i16_step=> ,
	i16_last_step=> );

CASE fb_state_entry.i16_next_step OF
(*=======================================================*)
	0:
		IF b_Execute THEN
			fb_state_entry.i16_next_step := 10;
		END_IF

(*=======================================================*)
	10:	(* Get Symbolinfo if necessary *)
		b_Busy := TRUE;
		IF str_SymInfo.idxGroup <> 0 AND s_SymbolName = s_SymbolNameOld THEN
			fb_state_entry.i16_next_step := 100;
		ELSE
			fb_state_entry.i16_next_step := 20;
		END_IF

(*=======================================================*)
	20:	(* Read Symbolinfo *)
		fb_read_symbolinfo.START := TRUE;
		IF fb_read_symbolinfo.BUSY THEN
			fb_state_entry.i16_next_step := 30;
		END_IF

(*=======================================================*)
	30:	(* Done or Error *)
		IF NOT fb_read_symbolinfo.BUSY THEN
			IF NOT fb_read_symbolinfo.ERR THEN
				fb_read_symbolinfo.START := FALSE;
				s_SymbolNameOld := s_SymbolName;
				fb_state_entry.i16_next_step := 100;
			ELSE
				b_Error := TRUE;
				b_ErrorID := fb_read_symbolinfo.ERRID;
				fb_state_entry.i16_next_step := 1000;
			END_IF
		END_IF

(*=======================================================*)
	100:	(* Read Symbol-Data *)
			fb_ads_write.WRITE := TRUE;
			IF fb_ads_write.BUSY THEN
				fb_state_entry.i16_next_step := 110;
			END_IF

(*=======================================================*)
	110:	(* Read is Busy *)
		IF NOT fb_ads_write.BUSY THEN
			IF NOT fb_ads_write.ERR THEN
				fb_ads_write.WRITE := FALSE;
				b_Done := TRUE;
				b_Busy := FALSE;
				fb_state_entry.i16_next_step := 120;
			ELSE
				b_Error := TRUE;
				b_ErrorID := fb_ads_write.ERRID;
				fb_state_entry.i16_next_step := 1000;
			END_IF
		END_IF

(*=======================================================*)
	120:	(* Read erfolgreich abgeschlossen *)
		IF NOT b_Execute THEN
			b_Done := FALSE;
			b_Busy := FALSE;
			fb_state_entry.i16_next_step := 0;
		END_IF;

(*=======================================================*)
	1000:	(* Fehler *)
		fb_read_symbolinfo.START := FALSE;
		fb_ads_write.WRITE := FALSE;

		IF b_Reset THEN
			fb_state_entry.i16_next_step := 0;
			b_Done := FALSE;
			b_Busy := FALSE;
			b_Error := FALSE;
			b_ErrorID := 0;
		END_IF

END_CASE

fb_state_entry(
	i16_next_step:= , 
	i16_pos:= 2,
	s_debugtext:= ,
	E=> , 
	X=> ,
	i16_step=> ,
	i16_last_step=> );

fb_read_symbolinfo(
	NETID:= AmsNetId,
	PORT:= Port,
	SYMNAME:= s_SymbolName,
	START:= , 
	TMOUT:= DEFAULT_ADS_TIMEOUT,
	BUSY=> , 
	ERR=> , 
	ERRID=> , 
	SYMINFO=> str_SymInfo);

fb_ads_write(
	NETID:= AmsNetId,
	PORT:= Port,
	IDXGRP:= str_SymInfo.idxGroup,
	IDXOFFS:= str_SymInfo.idxOffset,
	LEN:= str_SymInfo.byteSize,
	SRCADDR:= dw_SourceAdr,
	WRITE:= ,
	TMOUT:= DEFAULT_ADS_TIMEOUT,
	BUSY=> , 
	ERR=> , 
	ERRID=> );
END_FUNCTION_BLOCK

(* POU EPT Lib/Funktionsbausteine/ST_AnalogIn, ST *)
FUNCTION_BLOCK ST_AnalogIn
VAR_INPUT
	t_verzoegerung				: TIME;
	st_config						: struct_config;
END_VAR
VAR_OUTPUT
END_VAR
VAR
	b_error						: BOOL := FALSE;
	e_i16_sensor_delayed_value	: INT := 0;
	i16_anzeigewert_max			: INT := 16#7FFF;
	i16_anzeigewert_min			: INT := 16#0000;
	r_offset_skalierung			: INT := 16#0000;
	r_gain_skalierung				: INT := 16#0000;
	fb_abfragetakt				: ST_Blinker;
	fb_r_trig_abfragetakt			: R_TRIG;
	sm_overrange				: BOOL := FALSE;
	sm_underrange				: BOOL := FALSE;
	sm_limit1						: BOOL := FALSE;
	sm_limit2						: BOOL := FALSE;
	sm_error						: BOOL := FALSE;
	st_sensor					AT %I* :struct_analog_in;
END_VAR
(* Aufbereitung und Skalierung eines analogen Sensorwertes *)
i16_anzeigewert_max := 16#7FFF;

(* Verzögerte Abfrage des Analogwertes *)
fb_abfragetakt(
	b_start:= TRUE,
	 t_taktzeit_on:= t_verzoegerung,
	 t_taktzeit_off:= t_verzoegerung,
	b_blinker_out=> );

fb_r_trig_abfragetakt(CLK:= fb_abfragetakt.b_blinker_out, Q=> );

IF fb_r_trig_abfragetakt.Q THEN
	e_i16_sensor_delayed_value := st_sensor.e_i16_value;
END_IF

(* Fehlermeldungen der Analogkarte *)
sm_overrange := st_sensor.e_b_status_overrange;
sm_underrange := st_sensor.e_b_status_underrange;
sm_limit1	:= BYTE_TO_BOOL (st_sensor.e_by_status_limit1);
sm_limit2	 := BYTE_TO_BOOL (st_sensor.e_by_status_limit2);
sm_error	:= st_sensor.e_b_status_error;

b_error := sm_overrange OR sm_underrange OR sm_limit1 OR sm_limit2 OR sm_error;

IF st_config.b_config_fertig THEN
	(* Fehlermeldungen und Betriebsmeldungen ab dem Startindex in die globalen Meldungsarrays schreiben *)
	garr_stoermeldungen[st_config.i16_meld_startindex + 0] := sm_overrange;
	garr_stoermeldungen[st_config.i16_meld_startindex + 1] := sm_underrange;
	garr_stoermeldungen[st_config.i16_meld_startindex + 2] := sm_limit1;
	garr_stoermeldungen[st_config.i16_meld_startindex + 3] := sm_limit2;
	garr_stoermeldungen[st_config.i16_meld_startindex + 4] := sm_error;
	garr_stoermeldungen[st_config.i16_meld_startindex + 5] := FALSE;
	garr_stoermeldungen[st_config.i16_meld_startindex + 6] := FALSE;
	garr_stoermeldungen[st_config.i16_meld_startindex + 7] := FALSE;
	garr_stoermeldungen[st_config.i16_meld_startindex + 8] := FALSE;
	garr_stoermeldungen[st_config.i16_meld_startindex + 9] := FALSE;
	garr_stoermeldungen[st_config.i16_meld_startindex + 10] := FALSE;
	garr_stoermeldungen[st_config.i16_meld_startindex + 11] := FALSE;
	garr_stoermeldungen[st_config.i16_meld_startindex + 12] := FALSE;
	garr_stoermeldungen[st_config.i16_meld_startindex + 13] := FALSE;
	garr_stoermeldungen[st_config.i16_meld_startindex + 14] := FALSE;
	garr_stoermeldungen[st_config.i16_meld_startindex + 15] := FALSE;
	garr_stoermeldungen[st_config.i16_meld_startindex + 16] := FALSE;
	garr_stoermeldungen[st_config.i16_meld_startindex + 17] := FALSE;
	garr_stoermeldungen[st_config.i16_meld_startindex + 18] := FALSE;
	garr_stoermeldungen[st_config.i16_meld_startindex + 19] := FALSE;
	
	garr_betriebsmeldungen[st_config.i16_meld_startindex + 0] := FALSE;
	garr_betriebsmeldungen[st_config.i16_meld_startindex + 1] := FALSE;
	garr_betriebsmeldungen[st_config.i16_meld_startindex + 2] := FALSE;
	garr_betriebsmeldungen[st_config.i16_meld_startindex + 3] := FALSE;
	garr_betriebsmeldungen[st_config.i16_meld_startindex + 4] := FALSE;
	garr_betriebsmeldungen[st_config.i16_meld_startindex + 5] := FALSE;
	garr_betriebsmeldungen[st_config.i16_meld_startindex + 6] := FALSE;
	garr_betriebsmeldungen[st_config.i16_meld_startindex + 7] := FALSE;
	garr_betriebsmeldungen[st_config.i16_meld_startindex + 8] := FALSE;
	garr_betriebsmeldungen[st_config.i16_meld_startindex + 9] := FALSE;
	garr_betriebsmeldungen[st_config.i16_meld_startindex + 10] := FALSE;
	garr_betriebsmeldungen[st_config.i16_meld_startindex + 11] := FALSE;
	garr_betriebsmeldungen[st_config.i16_meld_startindex + 12] := FALSE;
	garr_betriebsmeldungen[st_config.i16_meld_startindex + 13] := FALSE;
	garr_betriebsmeldungen[st_config.i16_meld_startindex + 14] := FALSE;
	garr_betriebsmeldungen[st_config.i16_meld_startindex + 15] := FALSE;
	garr_betriebsmeldungen[st_config.i16_meld_startindex + 16] := FALSE;
	garr_betriebsmeldungen[st_config.i16_meld_startindex + 17] := FALSE;
	garr_betriebsmeldungen[st_config.i16_meld_startindex + 18] := FALSE;
	garr_betriebsmeldungen[st_config.i16_meld_startindex + 19] := FALSE;
END_IF
END_FUNCTION_BLOCK

(* POU EPT Lib/Funktionsbausteine/ST_AnalogOut, ST *)
FUNCTION_BLOCK ST_AnalogOut
VAR_INPUT
	r_digital_in					: REAL;
	st_config						: struct_config;
END_VAR
VAR_OUTPUT
END_VAR
VAR
	b_error						: BOOL := FALSE;
	i16_ausgabewert_max			: INT := 16#7FFF;
	i16_ausgabewert_min			: INT := 16#0;
	i16_offset_skalierung			: INT := 16#0;
	i16_gain_skalierung			: INT := 16#CCC;
	i16_analogwert				: INT := 0;
	sm_error						: BOOL := FALSE;
	i16_analog_out				AT %Q* : INT;
END_VAR
(* ===Ausgabe eines analogen Sollwertes an einen Aktor=== *)
(* Die Kalibrierung der Geraden sollte hier nicht geändert werden!
Der Ausgabe wert ist vom Format INT, somit wurde kalibriert auf den maximalen Endwert von 7FFF mit der Steigung CCC.
Der Offset dient zum Verschieben der Geraden, wenn bei Eingangswert 0 kein Analogwert von 0 erreicht wird. *)

IF st_config.b_station_aktiv THEN
	(* Skalieren des Analogwertes und Ausgabe an die Karte: y = gain*wert + offset *)
	i16_analogwert := REAL_TO_INT(INT_TO_REAL(i16_gain_skalierung) * r_digital_in + INT_TO_REAL(i16_offset_skalierung));
	
	IF i16_analogwert < i16_ausgabewert_min THEN
		i16_analog_out := i16_ausgabewert_min;
		b_error := TRUE;
	ELSIF i16_analogwert > i16_ausgabewert_max THEN
		i16_analog_out := i16_ausgabewert_max;
		b_error := TRUE;
	ELSE
		i16_analog_out := i16_analogwert;
		b_error := FALSE;
	END_IF
ELSE
	i16_analog_out := 0;
	b_error := FALSE;
END_IF

(* Fehlermeldung Bereich *)
sm_error := b_error;

IF st_config.b_config_fertig THEN
	(* Fehlermeldungen und Betriebsmeldungen ab dem Startindex in die globalen Meldungsarrays schreiben *)
	garr_stoermeldungen[st_config.i16_meld_startindex + 0] := sm_error;
	garr_stoermeldungen[st_config.i16_meld_startindex + 1] := FALSE;
	garr_stoermeldungen[st_config.i16_meld_startindex + 2] := FALSE;
	garr_stoermeldungen[st_config.i16_meld_startindex + 3] := FALSE;
	garr_stoermeldungen[st_config.i16_meld_startindex + 4] := FALSE;
	garr_stoermeldungen[st_config.i16_meld_startindex + 5] := FALSE;
	garr_stoermeldungen[st_config.i16_meld_startindex + 6] := FALSE;
	garr_stoermeldungen[st_config.i16_meld_startindex + 7] := FALSE;
	garr_stoermeldungen[st_config.i16_meld_startindex + 8] := FALSE;
	garr_stoermeldungen[st_config.i16_meld_startindex + 9] := FALSE;
	garr_stoermeldungen[st_config.i16_meld_startindex + 10] := FALSE;
	garr_stoermeldungen[st_config.i16_meld_startindex + 11] := FALSE;
	garr_stoermeldungen[st_config.i16_meld_startindex + 12] := FALSE;
	garr_stoermeldungen[st_config.i16_meld_startindex + 13] := FALSE;
	garr_stoermeldungen[st_config.i16_meld_startindex + 14] := FALSE;
	garr_stoermeldungen[st_config.i16_meld_startindex + 15] := FALSE;
	garr_stoermeldungen[st_config.i16_meld_startindex + 16] := FALSE;
	garr_stoermeldungen[st_config.i16_meld_startindex + 17] := FALSE;
	garr_stoermeldungen[st_config.i16_meld_startindex + 18] := FALSE;
	garr_stoermeldungen[st_config.i16_meld_startindex + 19] := FALSE;
	
	garr_betriebsmeldungen[st_config.i16_meld_startindex + 0] := FALSE;
	garr_betriebsmeldungen[st_config.i16_meld_startindex + 1] := FALSE;
	garr_betriebsmeldungen[st_config.i16_meld_startindex + 2] := FALSE;
	garr_betriebsmeldungen[st_config.i16_meld_startindex + 3] := FALSE;
	garr_betriebsmeldungen[st_config.i16_meld_startindex + 4] := FALSE;
	garr_betriebsmeldungen[st_config.i16_meld_startindex + 5] := FALSE;
	garr_betriebsmeldungen[st_config.i16_meld_startindex + 6] := FALSE;
	garr_betriebsmeldungen[st_config.i16_meld_startindex + 7] := FALSE;
	garr_betriebsmeldungen[st_config.i16_meld_startindex + 8] := FALSE;
	garr_betriebsmeldungen[st_config.i16_meld_startindex + 9] := FALSE;
	garr_betriebsmeldungen[st_config.i16_meld_startindex + 10] := FALSE;
	garr_betriebsmeldungen[st_config.i16_meld_startindex + 11] := FALSE;
	garr_betriebsmeldungen[st_config.i16_meld_startindex + 12] := FALSE;
	garr_betriebsmeldungen[st_config.i16_meld_startindex + 13] := FALSE;
	garr_betriebsmeldungen[st_config.i16_meld_startindex + 14] := FALSE;
	garr_betriebsmeldungen[st_config.i16_meld_startindex + 15] := FALSE;
	garr_betriebsmeldungen[st_config.i16_meld_startindex + 16] := FALSE;
	garr_betriebsmeldungen[st_config.i16_meld_startindex + 17] := FALSE;
	garr_betriebsmeldungen[st_config.i16_meld_startindex + 18] := FALSE;
	garr_betriebsmeldungen[st_config.i16_meld_startindex + 19] := FALSE;
END_IF
END_FUNCTION_BLOCK

(* POU EPT Lib/Serielle Kommunikation/ST_BalluffTagReader, ST *)
FUNCTION_BLOCK ST_BalluffTagReader
VAR_INPUT
	st_config						: struct_config;
	i16_addresse					: INT := 0;
	i16_anzahl_byte				: INT := 0;
	s_schreib_daten				: ARRAY [0..100] OF BYTE;
	st_ctrl_in						: struct_ctrl_in;
END_VAR
VAR_OUTPUT
	s_lese_daten					: ARRAY [0..100] OF BYTE;
	s_transp_serial_number		: STRING;
	st_ctrl_out					: struct_ctrl_out;
END_VAR
VAR
	fb_ton_wz					: TON;
	fb_ton_uez					: TON;
	fb_ton_quitt					: TON;
	fb_r_trig_lesen				: R_TRIG;
	fb_r_trig_schreiben			: R_TRIG;
	t_wz							: TIME := t#0ms;
	fb_state_entry					: ST_StateEntry;
	fb_r_trig_ibn_lesen			: R_TRIG;
	fb_r_trig_ibn_schreiben			: R_TRIG;
	fb_ton_ibn_lesen				: TON;
	fb_ton_ibn_schreiben			: TON;
	b_ibn_lesen					: BOOL := FALSE;
	b_ibn_schreiben				: BOOL := FALSE;
	sm_fehler_rfid_reader			: BOOL := FALSE;
	sm_kein_tag_erkannt			: BOOL := FALSE;

	(* Puffer für RS232*)
	RxBuffer						:ComBuffer;
	TxBuffer						:ComBuffer;
	EL6ComInData AT %I* 			:EL6inData22B;
	EL6ComOutData AT %Q*  		:EL6outData22B;
	fb_serial_line					: SerialLineControl ;

	(* RFID *)
	fb_RFID_Reader				: FB_RFIDReader;
	st_access_data				: ST_RFID_AccessData;
	eErrCodeRcv					: E_RFID_ErrCodeRcv_Balluff;

	e_tag_im_aktionsfeld			AT %I* : BOOL;
END_VAR
(* Zeiten *)
fb_ton_wz(IN:= , PT:= , Q=>  , ET=> );
fb_ton_uez(IN:= , PT:= , Q=>  , ET=> );
fb_ton_quitt(IN:= , PT:= t#100ms, Q=> , ET=> );
fb_r_trig_lesen(CLK:= st_ctrl_in.b_start_lesen, Q=> );
fb_r_trig_schreiben(CLK:= st_ctrl_in.b_start_schreiben, Q=> );

(* Inbetriebnahme *)
fb_r_trig_ibn_lesen(CLK:= b_ibn_lesen, Q=> );
fb_r_trig_ibn_schreiben(CLK:= b_ibn_schreiben, Q=> );
fb_ton_ibn_lesen(IN:= , PT:= t#1s, Q=> , ET=> );
fb_ton_ibn_schreiben(IN:= , PT:= t#1s, Q=> , ET=> );

IF fb_r_trig_ibn_lesen.Q THEN
	fb_ton_ibn_lesen.IN := TRUE;
ELSE
	IF fb_ton_ibn_lesen.Q THEN
		b_ibn_lesen := FALSE;
	 	fb_ton_ibn_lesen.IN := FALSE;
	END_IF
END_IF

IF fb_r_trig_ibn_schreiben.Q THEN
	fb_ton_ibn_schreiben.IN := TRUE;
ELSE
	IF fb_ton_ibn_schreiben.Q THEN
		b_ibn_schreiben := FALSE;
	 	fb_ton_ibn_schreiben.IN := FALSE;
	END_IF
END_IF


(* Toplevel *)(*
IF fb_state_entry.i16_next_step > INIT AND fb_state_entry.i16_next_step < FEHLER THEN
	IF fb_state_entry.i16_next_step < STOP THEN
		IF st_ctrl_in.b_stop THEN
			fb_state_entry.i16_next_step := STOP;
		END_IF
	END_IF
END_IF*)

(* ==================================Schrittkette================================ *)
fb_state_entry(
	i16_next_step:= ,
	i16_pos:= 1,
	s_debugtext:= ,
	E=> ,
	X=> , 
	i16_step=> ,
	i16_last_step=> );

CASE fb_state_entry.i16_step OF
(*=======================================================*)
	INIT_OBJ:
		fb_state_entry.i16_next_step := INIT;

(*=======================================================*)
	INIT:
		IF fb_state_entry.E THEN
			fb_ton_wz.IN := FALSE;
			fb_ton_uez.IN := FALSE;
			fb_ton_quitt.IN := FALSE;
			sm_fehler_rfid_reader := FALSE;
			sm_kein_tag_erkannt := FALSE;
			fb_RFID_Reader.bExecute := FALSE;
			st_ctrl_out.b_fehler := FALSE;
			st_ctrl_out.b_bereit := FALSE;
			st_ctrl_out.b_fertig := FALSE;
		END_IF

		(*-----------------------Weiterschaltbedingungen----------------------------*)
(*		IF st_ctrl_in.b_init THEN*)
			fb_state_entry.i16_next_step := 20;
(*		END_IF*)

(*=======================================================*)
	20:	(* Reset Reader *)
		IF fb_state_entry.E THEN
			fb_RFID_Reader.bExecute := TRUE;
			fb_RFID_Reader.eCommand := eRFC_ResetReader;
		END_IF
	
		(*-----------------------Weiterschaltbedingungen----------------------------*)
		IF fb_RFID_Reader.bBusy THEN
			fb_state_entry.i16_next_step := 30;
		END_IF

(*=======================================================*)
	30:

		(*-----------------------Weiterschaltbedingungen----------------------------*)
		IF NOT fb_RFID_Reader.bBusy THEN
			fb_RFID_Reader.bExecute := FALSE;
			IF fb_RFID_Reader.bResponseRcv THEN
				fb_state_entry.i16_next_step := BEREIT;
			ELSIF  fb_RFID_Reader.bError THEN
				eErrCodeRcv := fb_RFID_Reader.iErrorID;
				sm_fehler_rfid_reader := TRUE;
				fb_state_entry.i16_next_step := FEHLER;
			END_IF
		END_IF

(*=======================================================*)
	BEREIT:
		IF fb_state_entry.E THEN
			st_ctrl_out.b_bereit := TRUE;
			st_ctrl_out.b_fertig := TRUE;
		END_IF

		IF fb_r_trig_lesen.Q OR fb_r_trig_ibn_lesen.Q THEN
			st_ctrl_out.b_fertig := FALSE;
			fb_state_entry.i16_next_step := 200;
		ELSIF fb_r_trig_schreiben.Q OR fb_r_trig_ibn_schreiben.Q THEN
			st_ctrl_out.b_fertig := FALSE;
			fb_state_entry.i16_next_step := 300;
		END_IF

(*=======================================================*)
	200: (* Abfrage, ob sich ein Tag im Aktionsfeld befindet, damit gelesen werden kann. *)
		IF fb_state_entry.E THEN
			fb_ton_uez.PT := t#1s;
			fb_ton_uez.IN := TRUE;
		END_IF

		(*-----------------------Weiterschaltbedingungen----------------------------*)
		IF e_tag_im_aktionsfeld THEN
			fb_ton_uez.IN := FALSE;
			fb_state_entry.i16_next_step := 210;
		ELSIF fb_ton_uez.Q THEN
			sm_kein_tag_erkannt := TRUE;
			fb_state_entry.i16_next_step := FEHLER;
		END_IF

(*=======================================================*)
	210: (* Start Lesen *)
		(* Vorbereiten Lesen *)
		IF fb_state_entry.E THEN
			fb_RFID_Reader.bExecute := TRUE;
			fb_RFID_Reader.eCommand := eRFC_ReadBlock;

			(* Datasize = blockCount * BlockSize *)
			st_access_data.iDataSize := i16_anzahl_byte;
			st_access_data.iBlockCount := i16_anzahl_byte;
			st_access_data.iBlockSize := 1;
			st_access_data.iStartBlock := i16_addresse;

			MEMSET(ADR(s_lese_daten), 0 , SIZEOF(s_lese_daten) );
			st_access_data.pData := ADR(s_lese_daten);
		END_IF

		(*-----------------------Weiterschaltbedingungen----------------------------*)
		IF fb_RFID_Reader.bBusy THEN
			fb_state_entry.i16_next_step := 220;
		END_IF

(*=======================================================*)
	220:	(* Fertig Lesen *)

		(*-----------------------Weiterschaltbedingungen----------------------------*)
		IF NOT fb_RFID_Reader.bBusy THEN
			fb_RFID_Reader.bExecute := FALSE;
			IF fb_RFID_Reader.bResponseRcv THEN
				fb_state_entry.i16_next_step := BEREIT;
			ELSIF  fb_RFID_Reader.bError THEN
				eErrCodeRcv := fb_RFID_Reader.iErrorID;
				sm_fehler_rfid_reader := TRUE;
				fb_state_entry.i16_next_step := FEHLER;
			END_IF
		END_IF

(*=======================================================*)
	300: (* Abfrage, ob sich ein Tag im Aktionsfeld befindet, damit geschrieben werden kann. *)
		IF fb_state_entry.E THEN
			fb_ton_uez.PT := t#1s;
			fb_ton_uez.IN := TRUE;
		END_IF

		(*-----------------------Weiterschaltbedingungen----------------------------*)
		IF e_tag_im_aktionsfeld THEN
			fb_ton_uez.IN := FALSE;
			fb_state_entry.i16_next_step := 310;
		ELSIF fb_ton_uez.Q THEN
			sm_kein_tag_erkannt := TRUE;
			fb_state_entry.i16_next_step := FEHLER;
		END_IF

(*=======================================================*)
	310: (* Start Schreiben *)
		(* Vorbereiten Schreiben *)
		IF fb_state_entry.E THEN
			fb_RFID_Reader.bExecute := TRUE;
			fb_RFID_Reader.eCommand := eRFC_WriteBlock;

			(* Datasize = blockCount * BlockSize *)
			st_access_data.iDataSize := i16_anzahl_byte;
			st_access_data.iBlockCount := i16_anzahl_byte;
			st_access_data.iBlockSize := 1;
			st_access_data.iStartBlock := i16_addresse;

			st_access_data.pData := ADR(s_schreib_daten);
		END_IF

		(*-----------------------Weiterschaltbedingungen----------------------------*)
		IF fb_RFID_Reader.bBusy THEN
			fb_state_entry.i16_next_step := 320;
		END_IF

(*=======================================================*)
	320:	(* Fertig Schreiben *)

		(*-----------------------Weiterschaltbedingungen----------------------------*)
		IF NOT fb_RFID_Reader.bBusy THEN
			fb_RFID_Reader.bExecute := FALSE;
			IF fb_RFID_Reader.bResponseRcv THEN
				fb_state_entry.i16_next_step := BEREIT;
			ELSIF  fb_RFID_Reader.bError THEN
				eErrCodeRcv := fb_RFID_Reader.iErrorID;
				sm_fehler_rfid_reader := TRUE;
				fb_state_entry.i16_next_step := FEHLER;
			END_IF
		END_IF

(*=======================================================*)
	FEHLER:
		IF fb_state_entry.E THEN
			fb_RFID_Reader.bExecute := FALSE;
			st_ctrl_out.b_fehler := TRUE;
			fb_ton_quitt.IN := FALSE;
		END_IF

		(*-----------------------Weiterschaltbedingungen----------------------------*)
		IF st_ctrl_in.b_quitt AND NOT fb_state_entry.E THEN
			st_ctrl_out.b_fehler := FALSE;
			fb_ton_quitt.IN := TRUE;
		END_IF

